   1:  PR[91,3] = PR[90,3] + 136.116;
   1:L PR[91] R[100]mm/sec CNT100;
   1:  PR[91,1] = PR[90,1] + 83.828;
   1:  PR[91,2] = PR[90,2] + 8.492;
   1:  PR[91,3] = PR[90,3] + 136.123;
   1:L PR[91] R[100]mm/sec CNT100;
   1:  PR[91,1] = PR[90,1] + 81.539;
   1:  PR[91,2] = PR[90,2] + 13.617;
   1:  PR[91,3] = PR[90,3] + 136.131;
   1:L PR[91] R[100]mm/sec CNT100;
   1:  PR[91,1] = PR[90,1] + 80.801;
   1:  PR[91,2] = PR[90,2] + 14.808;
   1:  PR[91,3] = PR[90,3] + 136.163;
   1:L PR[91] R[100]mm/sec CNT100;
   1:  PR[91,1] = PR[90,1] + 75.916;
   1:  PR[91,2] = PR[90,2] + 20.688;
   1:  PR[91,3] = PR[90,3] + 136.171;
   1:L PR[91] R[100]mm/sec CNT100;
   1:  PR[91,1] = PR[90,1] + 74.686;
   1:  PR[91,2] = PR[90,2] + 21.792;
   1:  PR[91,3] = PR[90,3] + 136.214;
   1:L PR[91] R[100]mm/sec CNT100;
   1:  PR[91,1] = PR[90,1] + 72.953;
   1:  PR[91,2] = PR[90,2] + 22.987;
   1:  PR[91,3] = PR[90,3] + 136.223;
   1:L PR[91] R[100]mm/sec CNT100;
   1:  PR[91,1] = PR[90,1] + 67.912;
   1:  PR[91,2] = PR[90,2] + 26.567;
   1:  PR[91,3] = PR[90,3] + 136.235;
   1:L PR[91] R[100]mm/sec CNT100;
   1:  PR[91,1] = PR[90,1] + 66.099;
   1:  PR[91,2] = PR[90,2] + 27.495;
   1:  PR[91,3] = PR[90,3] + 136.270;
   1:L PR[91] R[100]mm/sec CNT100;
   1:  PR[91,1] = PR[90,1] + 63.634;
   1:  PR[91,2] = PR[90,2] + 28.417;
   1:  PR[91,3] = PR[90,3] + 136.281;
   1:L PR[91] R[100]mm/sec CNT100;
   1:  PR[91,1] = PR[90,1] + 57.996;
   1:  PR[91,2] = PR[90,2] + 30.575;
   1:  PR[91,3] = PR[90,3] + 136.296;
   1:L PR[91] R[100]mm/sec CNT100;
   1:  PR[91,1] = PR[90,1] + 55.467;
   1:  PR[91,2] = PR[90,2] + 31.181;
   1:  PR[91,3] = PR[90,3] + 136.330;
   1:L PR[91] R[100]mm/sec CNT100;
   1:  PR[91,1] = PR[90,1] + 52.680;
   1:  PR[91,2] = PR[90,2] + 31.695;
   1:  PR[91,3] = PR[90,3] + 136.345;
   1:L PR[91] R[100]mm/sec CNT100;
   1:  PR[91,1] = PR[90,1] + 49.741;
   1:  PR[91,2] = PR[90,2] + 32.053;
   1:  PR[91,3] = PR[90,3] + 136.361;
   1:L PR[91] R[100]mm/sec CNT100;
   1:  PR[91,1] = PR[90,1] + 47.228;
   1:  PR[91,2] = PR[90,2] + 32.206;
   1:  PR[91,3] = PR[90,3] + 136.378;
   1:L PR[91] R[100]mm/sec CNT100;
   1:  PR[91,1] = PR[90,1] + 43.917;
   1:  PR[91,2] = PR[90,2] + 32.236;
   1:  PR[91,3] = PR[90,3] + 136.392;
   1:L PR[91] R[100]mm/sec CNT100;
   1:  PR[91,1] = PR[90,1] + 41.866;
   1:  PR[91,2] = PR[90,2] + 32.111;
   1:  PR[91,3] = PR[90,3] + 136.411;
   1:L PR[91] R[100]mm/sec CNT100;
   1:  PR[91,1] = PR[90,1] + 38.413;
   1:  PR[91,2] = PR[90,2] + 31.768;
   1:  PR[91,3] = PR[90,3] + 136.422;
   1:L PR[91] R[100]mm/sec CNT100;
   1:  PR[91,1] = PR[90,1] + 36.971;
   1:  PR[91,2] = PR[90,2] + 31.502;
   1:  PR[91,3] = PR[90,3] + 136.442;
   1:L PR[91] R[100]mm/sec CNT100;
   1:  PR[91,1] = PR[90,1] + 33.194;
   1:  PR[91,2] = PR[90,2] + 30.719;
   1:  PR[91,3] = PR[90,3] + 136.450;
   1:L PR[91] R[100]mm/sec CNT100;
   1:  PR[91,1] = PR[90,1] + 28.411;
   1:  PR[91,2] = PR[90,2] + 29.184;
   1:  PR[91,3] = PR[90,3] + 136.472;
   1:L PR[91] R[100]mm/sec CNT100;
   1:  PR[91,1] = PR[90,1] + 24.182;
   1:  PR[91,2] = PR[90,2] + 27.259;
   1:  PR[91,3] = PR[90,3] + 136.500;
   1:L PR[91] R[100]mm/sec CNT100;
   1:  PR[91,1] = PR[90,1] + 19.400;
   1:  PR[91,2] = PR[90,2] + 24.371;
   1:  PR[91,3] = PR[90,3] + 136.527;
   1:L PR[91] R[100]mm/sec CNT100;
   1:  PR[91,1] = PR[90,1] + 18.294;
   1:  PR[91,2] = PR[90,2] + 23.512;
   1:  PR[91,3] = PR[90,3] + 136.558;
   1:L PR[91] R[100]mm/sec CNT100;
   1:  PR[91,1] = PR[90,1] + 14.337;
   1:  PR[91,2] = PR[90,2] + 20.137;
   1:  PR[91,3] = PR[90,3] + 136.566;
   1:L PR[91] R[100]mm/sec CNT100;
   1:  PR[91,1] = PR[90,1] + 10.437;
   1:  PR[91,2] = PR[90,2] + 15.629;
   1:  PR[91,3] = PR[90,3] + 136.595;
   1:L PR[91] R[100]mm/sec CNT100;
   1:  PR[91,1] = PR[90,1] + 8.817;
   1:  PR[91,2] = PR[90,2] + 12.942;
   1:  PR[91,3] = PR[90,3] + 136.629;
   1:L PR[91] R[100]mm/sec CNT100;
   1:  PR[91,1] = PR[90,1] + 7.454;
   1:  PR[91,2] = PR[90,2] + 10.581;
   1:  PR[91,3] = PR[90,3] + 136.647;
   1:L PR[91] R[100]mm/sec CNT100;
   1:  PR[91,1] = PR[90,1] + 5.830;
   1:  PR[91,2] = PR[90,2] + 5.883;
   1:  PR[91,3] = PR[90,3] + 136.662;
   1:L PR[91] R[100]mm/sec CNT100;
   1:  PR[91,1] = PR[90,1] + 5.557;
   1:  PR[91,2] = PR[90,2] + 5.060;
   1:  PR[91,3] = PR[90,3] + 136.690;
   1:L PR[91] R[100]mm/sec CNT100;
   1:  PR[91] = PR[90];
   1:  PR[91,1] = PR[90,1] + 6.034;
   1:  PR[91,2] = PR[90,2] + 1.066;
   1:  PR[91,3] = PR[90,3] + 137.995;
   1:L PR[91] R[100]mm/sec CNT100;
   1:  PR[91,1] = PR[90,1] + 5.903;
   1:  PR[91,2] = PR[90,2] + -0.687;
   1:  PR[91,3] = PR[90,3] + 136.717;
   1:L PR[91] R[100]mm/sec CNT100;
   1:  PR[91,1] = PR[90,1] + 6.070;
   1:  PR[91,2] = PR[90,2] + -2.112;
   1:  PR[91,3] = PR[90,3] + 136.727;
   1:L PR[91] R[100]mm/sec CNT100;
   1:  PR[91,1] = PR[90,1] + 6.290;
   1:  PR[91,2] = PR[90,2] + -4.587;
   1:  PR[91,3] = PR[90,3] + 136.735;
   1:L PR[91] R[100]mm/sec CNT100;
   1:  PR[91,1] = PR[90,1] + 6.492;
   1:  PR[91,2] = PR[90,2] + -6.475;
   1:  PR[91,3] = PR[90,3] + 136.749;
   1:L PR[91] R[100]mm/sec CNT100;
   1:  PR[91,1] = PR[90,1] + 7.257;
   1:  PR[91,2] = PR[90,2] + -8.786;
   1:  PR[91,3] = PR[90,3] + 136.760;
   1:L PR[91] R[100]mm/sec CNT100;
   1:  PR[91,1] = PR[90,1] + 8.349;
   1:  PR[91,2] = PR[90,2] + -11.947;
   1:  PR[91,3] = PR[90,3] + 136.774;
   1:L PR[91] R[100]mm/sec CNT100;
   1:  PR[91,1] = PR[90,1] + 10.575;
   1:  PR[91,2] = PR[90,2] + -15.804;
   1:  PR[91,3] = PR[90,3] + 136.793;
   1:L PR[91] R[100]mm/sec CNT100;
   1:  PR[91,1] = PR[90,1] + 11.282;
   1:  PR[91,2] = PR[90,2] + -16.976;
   1:  PR[91,3] = PR[90,3] + 136.818;
   1:L PR[91] R[100]mm/sec CNT100;
   1:  PR[91,1] = PR[90,1] + 13.229;
   1:  PR[91,2] = PR[90,2] + -19.231;
   1:  PR[91,3] = PR[90,3] + 136.826;
   1:L PR[91] R[100]mm/sec CNT100;
   1:  PR[91,1] = PR[90,1] + 15.024;
   1:  PR[91,2] = PR[90,2] + -21.414;
   1:  PR[91,3] = PR[90,3] + 136.843;
   1:L PR[91] R[100]mm/sec CNT100;
   1:  PR[91,1] = PR[90,1] + 15.491;
   1:  PR[91,2] = PR[90,2] + -21.879;
   1:  PR[91,3] = PR[90,3] + 136.858;
   1:L PR[91] R[100]mm/sec CNT100;
   1:  PR[91,1] = PR[90,1] + 18.681;
   1:  PR[91,2] = PR[90,2] + -24.609;
   1:  PR[91,3] = PR[90,3] + 136.862;
   1:L PR[91] R[100]mm/sec CNT100;
   1:  PR[91,1] = PR[90,1] + 20.378;
   1:  PR[91,2] = PR[90,2] + -25.927;
   1:  PR[91,3] = PR[90,3] + 136.886;
   1:L PR[91] R[100]mm/sec CNT100;
   1:  PR[91,1] = PR[90,1] + 22.117;
   1:  PR[91,2] = PR[90,2] + -26.965;
   1:  PR[91,3] = PR[90,3] + 136.898;
   1:L PR[91] R[100]mm/sec CNT100;
   1:  PR[91,1] = PR[90,1] + 24.901;
   1:  PR[91,2] = PR[90,2] + -28.668;
   1:  PR[91,3] = PR[90,3] + 136.909;
   1:L PR[91] R[100]mm/sec CNT100;
   1:  PR[91,1] = PR[90,1] + 28.747;
   1:  PR[91,2] = PR[90,2] + -30.406;
   1:  PR[91,3] = PR[90,3] + 136.928;
   1:L PR[91] R[100]mm/sec CNT100;
   1:  PR[91,1] = PR[90,1] + 31.797;
   1:  PR[91,2] = PR[90,2] + -31.291;
   1:  PR[91,3] = PR[90,3] + 136.952;
   1:L PR[91] R[100]mm/sec CNT100;
   1:  PR[91,1] = PR[90,1] + 34.180;
   1:  PR[91,2] = PR[90,2] + -32.203;
   1:  PR[91,3] = PR[90,3] + 136.970;
   1:L PR[91] R[100]mm/sec CNT100;
   1:  PR[91,1] = PR[90,1] + 37.512;
   1:  PR[91,2] = PR[90,2] + -32.893;
   1:  PR[91,3] = PR[90,3] + 136.984;
   1:L PR[91] R[100]mm/sec CNT100;
   1:  PR[91,1] = PR[90,1] + 39.398;
   1:  PR[91,2] = PR[90,2] + -33.241;
   1:  PR[91,3] = PR[90,3] + 137.003;
   1:L PR[91] R[100]mm/sec CNT100;
   1:  PR[91,1] = PR[90,1] + 42.493;
   1:  PR[91,2] = PR[90,2] + -33.549;
   1:  PR[91,3] = PR[90,3] + 137.014;
   1:L PR[91] R[100]mm/sec CNT100;
   1:  PR[91,1] = PR[90,1] + 44.945;
   1:  PR[91,2] = PR[90,2] + -33.699;
   1:  PR[91,3] = PR[90,3] + 137.032;
   1:L PR[91] R[100]mm/sec CNT100;
   1:  PR[91,1] = PR[90,1] + 47.912;
   1:  PR[91,2] = PR[90,2] + -33.672;
   1:  PR[91,3] = PR[90,3] + 137.046;
   1:L PR[91] R[100]mm/sec CNT100;
   1:  PR[91,1] = PR[90,1] + 50.781;
   1:  PR[91,2] = PR[90,2] + -33.496;
   1:  PR[91,3] = PR[90,3] + 137.062;
   1:L PR[91] R[100]mm/sec CNT100;
   1:  PR[91,1] = PR[90,1] + 53.413;
   1:  PR[91,2] = PR[90,2] + -33.175;
   1:  PR[91,3] = PR[90,3] + 137.079;
   1:L PR[91] R[100]mm/sec CNT100;
   1:  PR[91,1] = PR[90,1] + 56.507;
   1:  PR[91,2] = PR[90,2] + -32.604;
   1:  PR[91,3] = PR[90,3] + 137.094;
   1:L PR[91] R[100]mm/sec CNT100;
   1:  PR[91,1] = PR[90,1] + 58.774;
   1:  PR[91,2] = PR[90,2] + -32.061;
   1:  PR[91,3] = PR[90,3] + 137.111;
   1:L PR[91] R[100]mm/sec CNT100;
   1:  PR[91,1] = PR[90,1] + 60.594;
   1:  PR[91,2] = PR[90,2] + -31.384;
   1:  PR[91,3] = PR[90,3] + 137.124;
   1:L PR[91] R[100]mm/sec CNT100;
   1:  PR[91,1] = PR[90,1] + 67.110;
   1:  PR[91,2] = PR[90,2] + -28.889;
   1:  PR[91,3] = PR[90,3] + 137.135;
   1:L PR[91] R[100]mm/sec CNT100;
   1:  PR[91,1] = PR[90,1] + 68.740;
   1:  PR[91,2] = PR[90,2] + -28.055;
   1:  PR[91,3] = PR[90,3] + 137.175;
   1:L PR[91] R[100]mm/sec CNT100;
   1:  PR[91,1] = PR[90,1] + 70.080;
   1:  PR[91,2] = PR[90,2] + -27.134;
   1:  PR[91,3] = PR[90,3] + 137.185;
   1:L PR[91] R[100]mm/sec CNT100;
   1:  PR[91,1] = PR[90,1] + 75.649;
   1:  PR[91,2] = PR[90,2] + -23.178;
   1:  PR[91,3] = PR[90,3] + 137.194;
   1:L PR[91] R[100]mm/sec CNT100;
   1:  PR[91,1] = PR[90,1] + 76.745;
   1:  PR[91,2] = PR[90,2] + -22.194;
   1:  PR[91,3] = PR[90,3] + 137.233;
   1:L PR[91] R[100]mm/sec CNT100;
   1:  PR[91,1] = PR[90,1] + 81.726;
   1:  PR[91,2] = PR[90,2] + -16.195;
   1:  PR[91,3] = PR[90,3] + 137.241;
   1:L PR[91] R[100]mm/sec CNT100;
   1:  PR[91,1] = PR[90,1] + 82.365;
   1:  PR[91,2] = PR[90,2] + -15.164;
   1:  PR[91,3] = PR[90,3] + 137.285;
   1:L PR[91] R[100]mm/sec CNT100;
   1:  PR[91,1] = PR[90,1] + 82.859;
   1:  PR[91,2] = PR[90,2] + -13.996;
   1:  PR[91,3] = PR[90,3] + 137.292;
   1:L PR[91] R[100]mm/sec CNT100;
   1:  PR[91,1] = PR[90,1] + 85.287;
   1:  PR[91,2] = PR[90,2] + -8.560;
   1:  PR[91,3] = PR[90,3] + 137.299;
   1:L PR[91] R[100]mm/sec CNT100;
   1:  PR[91,1] = PR[90,1] + 85.539;
   1:  PR[91,2] = PR[90,2] + -7.546;
   1:  PR[91,3] = PR[90,3] + 137.333;
   1:L PR[91] R[100]mm/sec CNT100;
   1:  PR[91,1] = PR[90,1] + 85.641;
   1:  PR[91,2] = PR[90,2] + -6.296;
   1:  PR[91,3] = PR[90,3] + 137.339;
   1:L PR[91] R[100]mm/sec CNT100;
   1:  PR[91,1] = PR[90,1] + 86.439;
   1:  PR[91,2] = PR[90,2] + -0.670;
   1:  PR[91,3] = PR[90,3] + 137.346;
   1:L PR[91] R[100]mm/sec CNT100;
   1:  PR[91,1] = PR[90,1] + 86.350;
   1:  PR[91,2] = PR[90,2] + 0.412;
   1:  PR[91,3] = PR[90,3] + 137.378;
   1:L PR[91] R[100]mm/sec CNT100;
   1:  PR[91,1] = PR[90,1] + 85.554;
   1:  PR[91,2] = PR[90,2] + 6.030;
   1:  PR[91,3] = PR[90,3] + 137.384;
   1:L PR[91] R[100]mm/sec CNT100;
   1:  PR[91,1] = PR[90,1] + 85.282;
   1:  PR[91,2] = PR[90,2] + 7.121;
   1:  PR[91,3] = PR[90,3] + 137.416;
   1:L PR[91] R[100]mm/sec CNT100;
   1:  PR[91,1] = PR[90,1] + 84.781;
   1:  PR[91,2] = PR[90,2] + 8.302;
   1:  PR[91,3] = PR[90,3] + 137.422;
   1:L PR[91] R[100]mm/sec CNT100;
   1:  PR[91,1] = PR[90,1] + 82.374;
   1:  PR[91,2] = PR[90,2] + 13.690;
   1:  PR[91,3] = PR[90,3] + 137.430;
   1:L PR[91] R[100]mm/sec CNT100;
   1:  PR[91,1] = PR[90,1] + 81.725;
   1:  PR[91,2] = PR[90,2] + 14.738;
   1:  PR[91,3] = PR[90,3] + 137.463;
   1:L PR[91] R[100]mm/sec CNT100;
   1:  PR[91,1] = PR[90,1] + 76.743;
   1:  PR[91,2] = PR[90,2] + 20.737;
   1:  PR[91,3] = PR[90,3] + 137.470;
   1:L PR[91] R[100]mm/sec CNT100;
   1:  PR[91,1] = PR[90,1] + 75.657;
   1:  PR[91,2] = PR[90,2] + 21.711;
   1:  PR[91,3] = PR[90,3] + 137.514;
   1:L PR[91] R[100]mm/sec CNT100;
   1:  PR[91,1] = PR[90,1] + 74.107;
   1:  PR[91,2] = PR[90,2] + 22.780;
   1:  PR[91,3] = PR[90,3] + 137.522;
   1:L PR[91] R[100]mm/sec CNT100;
   1:  PR[91,1] = PR[90,1] + 68.723;
   1:  PR[91,2] = PR[90,2] + 26.605;
   1:  PR[91,3] = PR[90,3] + 137.533;
   1:L PR[91] R[100]mm/sec CNT100;
   1:  PR[91,1] = PR[90,1] + 67.114;
   1:  PR[91,2] = PR[90,2] + 27.428;
   1:  PR[91,3] = PR[90,3] + 137.570;
   1:L PR[91] R[100]mm/sec CNT100;
   1:  PR[91,1] = PR[90,1] + 64.907;
   1:  PR[91,2] = PR[90,2] + 28.253;
   1:  PR[91,3] = PR[90,3] + 137.580;
   1:L PR[91] R[100]mm/sec CNT100;
   1:  PR[91,1] = PR[90,1] + 58.762;
   1:  PR[91,2] = PR[90,2] + 30.605;
   1:  PR[91,3] = PR[90,3] + 137.594;
   1:L PR[91] R[100]mm/sec CNT100;
   1:  PR[91,1] = PR[90,1] + 56.504;
   1:  PR[91,2] = PR[90,2] + 31.146;
   1:  PR[91,3] = PR[90,3] + 137.631;
   1:L PR[91] R[100]mm/sec CNT100;
   1:  PR[91,1] = PR[90,1] + 53.410;
   1:  PR[91,2] = PR[90,2] + 31.717;
   1:  PR[91,3] = PR[90,3] + 137.644;
   1:L PR[91] R[100]mm/sec CNT100;
   1:  PR[91,1] = PR[90,1] + 50.778;
   1:  PR[91,2] = PR[90,2] + 32.037;
   1:  PR[91,3] = PR[90,3] + 137.662;
   1:L PR[91] R[100]mm/sec CNT100;
   1:  PR[91,1] = PR[90,1] + 47.909;
   1:  PR[91,2] = PR[90,2] + 32.213;
   1:  PR[91,3] = PR[90,3] + 137.677;
   1:L PR[91] R[100]mm/sec CNT100;
   1:  PR[91,1] = PR[90,1] + 44.943;
   1:  PR[91,2] = PR[90,2] + 32.240;
   1:  PR[91,3] = PR[90,3] + 137.693;
   1:L PR[91] R[100]mm/sec CNT100;
   1:  PR[91,1] = PR[90,1] + 42.490;
   1:  PR[91,2] = PR[90,2] + 32.090;
   1:  PR[91,3] = PR[90,3] + 137.710;
   1:L PR[91] R[100]mm/sec CNT100;
   1:  PR[91,1] = PR[90,1] + 39.396;
   1:  PR[91,2] = PR[90,2] + 31.782;
   1:  PR[91,3] = PR[90,3] + 137.724;
   1:L PR[91] R[100]mm/sec CNT100;
   1:  PR[91,1] = PR[90,1] + 37.510;
   1:  PR[91,2] = PR[90,2] + 31.434;
   1:  PR[91,3] = PR[90,3] + 137.741;
   1:L PR[91] R[100]mm/sec CNT100;
   1:  PR[91,1] = PR[90,1] + 34.124;
   1:  PR[91,2] = PR[90,2] + 30.732;
   1:  PR[91,3] = PR[90,3] + 137.752;
   1:L PR[91] R[100]mm/sec CNT100;
   1:  PR[91,1] = PR[90,1] + 29.707;
   1:  PR[91,2] = PR[90,2] + 29.318;
   1:  PR[91,3] = PR[90,3] + 137.771;
   1:L PR[91] R[100]mm/sec CNT100;
   1:  PR[91,1] = PR[90,1] + 26.882;
   1:  PR[91,2] = PR[90,2] + 28.114;
   1:  PR[91,3] = PR[90,3] + 137.798;
   1:L PR[91] R[100]mm/sec CNT100;
   1:  PR[91,1] = PR[90,1] + 24.902;
   1:  PR[91,2] = PR[90,2] + 27.210;
   1:  PR[91,3] = PR[90,3] + 137.815;
   1:L PR[91] R[100]mm/sec CNT100;
   1:  PR[91,1] = PR[90,1] + 20.385;
   1:  PR[91,2] = PR[90,2] + 24.473;
   1:  PR[91,3] = PR[90,3] + 137.827;
   1:L PR[91] R[100]mm/sec CNT100;
   1:  PR[91,1] = PR[90,1] + 18.684;
   1:  PR[91,2] = PR[90,2] + 23.151;
   1:  PR[91,3] = PR[90,3] + 137.857;
   1:L PR[91] R[100]mm/sec CNT100;
   1:  PR[91,1] = PR[90,1] + 15.494;
   1:  PR[91,2] = PR[90,2] + 20.423;
   1:  PR[91,3] = PR[90,3] + 137.869;
   1:L PR[91] R[100]mm/sec CNT100;
   1:  PR[91,1] = PR[90,1] + 15.026;
   1:  PR[91,2] = PR[90,2] + 19.958;
   1:  PR[91,3] = PR[90,3] + 137.893;
   1:L PR[91] R[100]mm/sec CNT100;
   1:  PR[91,1] = PR[90,1] + 13.229;
   1:  PR[91,2] = PR[90,2] + 17.772;
   1:  PR[91,3] = PR[90,3] + 137.897;
   1:L PR[91] R[100]mm/sec CNT100;
   1:  PR[91,1] = PR[90,1] + 11.284;
   1:  PR[91,2] = PR[90,2] + 15.520;
   1:  PR[91,3] = PR[90,3] + 137.913;
   1:L PR[91] R[100]mm/sec CNT100;
   1:  PR[91,1] = PR[90,1] + 10.578;
   1:  PR[91,2] = PR[90,2] + 14.349;
   1:  PR[91,3] = PR[90,3] + 137.929;
   1:L PR[91] R[100]mm/sec CNT100;
   1:  PR[91,1] = PR[90,1] + 8.351;
   1:  PR[91,2] = PR[90,2] + 10.491;
   1:  PR[91,3] = PR[90,3] + 137.937;
   1:L PR[91] R[100]mm/sec CNT100;
   1:  PR[91,1] = PR[90,1] + 7.258;
   1:  PR[91,2] = PR[90,2] + 7.330;
   1:  PR[91,3] = PR[90,3] + 137.962;
   1:L PR[91] R[100]mm/sec CNT100;
   1:  PR[91,1] = PR[90,1] + 6.489;
   1:  PR[91,2] = PR[90,2] + 5.009;
   1:  PR[91,3] = PR[90,3] + 137.981;
   1:L PR[91] R[100]mm/sec CNT100;
   1:  PR[91] = PR[90];
   1:  PR[91,1] = PR[90,1] + 7.128;
   1:  PR[91,2] = PR[90,2] + 2.420;
   1:  PR[91,3] = PR[90,3] + 139.295;
   1:L PR[91] R[100]mm/sec CNT100;
   1:  PR[91,1] = PR[90,1] + 6.959;
   1:  PR[91,2] = PR[90,2] + 0.156;
   1:  PR[91,3] = PR[90,3] + 138.009;
   1:L PR[91] R[100]mm/sec CNT100;
   1:  PR[91,1] = PR[90,1] + 6.863;
   1:  PR[91,2] = PR[90,2] + -0.747;
   1:  PR[91,3] = PR[90,3] + 138.022;
   1:L PR[91] R[100]mm/sec CNT100;
   1:  PR[91,1] = PR[90,1] + 7.088;
   1:  PR[91,2] = PR[90,2] + -3.281;
   1:  PR[91,3] = PR[90,3] + 138.027;
   1:L PR[91] R[100]mm/sec CNT100;
   1:  PR[91,1] = PR[90,1] + 7.424;
   1:  PR[91,2] = PR[90,2] + -6.424;
   1:  PR[91,3] = PR[90,3] + 138.042;
   1:L PR[91] R[100]mm/sec CNT100;
   1:  PR[91,1] = PR[90,1] + 8.684;
   1:  PR[91,2] = PR[90,2] + -10.233;
   1:  PR[91,3] = PR[90,3] + 138.060;
   1:L PR[91] R[100]mm/sec CNT100;
   1:  PR[91,1] = PR[90,1] + 9.246;
   1:  PR[91,2] = PR[90,2] + -11.859;
   1:  PR[91,3] = PR[90,3] + 138.082;
   1:L PR[91] R[100]mm/sec CNT100;
   1:  PR[91,1] = PR[90,1] + 12.150;
   1:  PR[91,2] = PR[90,2] + -16.909;
   1:  PR[91,3] = PR[90,3] + 138.092;
   1:L PR[91] R[100]mm/sec CNT100;
   1:  PR[91,1] = PR[90,1] + 15.624;
   1:  PR[91,2] = PR[90,2] + -21.142;
   1:  PR[91,3] = PR[90,3] + 138.125;
   1:L PR[91] R[100]mm/sec CNT100;
   1:  PR[91,1] = PR[90,1] + 16.758;
   1:  PR[91,2] = PR[90,2] + -22.269;
   1:  PR[91,3] = PR[90,3] + 138.156;
   1:L PR[91] R[100]mm/sec CNT100;
   1:  PR[91,1] = PR[90,1] + 19.070;
   1:  PR[91,2] = PR[90,2] + -24.247;
   1:  PR[91,3] = PR[90,3] + 138.165;
   1:L PR[91] R[100]mm/sec CNT100;
   1:  PR[91,1] = PR[90,1] + 21.369;
   1:  PR[91,2] = PR[90,2] + -26.033;
   1:  PR[91,3] = PR[90,3] + 138.182;
   1:L PR[91] R[100]mm/sec CNT100;
   1:  PR[91,1] = PR[90,1] + 25.631;
   1:  PR[91,2] = PR[90,2] + -28.617;
   1:  PR[91,3] = PR[90,3] + 138.198;
   1:L PR[91] R[100]mm/sec CNT100;
   1:  PR[91,1] = PR[90,1] + 29.090;
   1:  PR[91,2] = PR[90,2] + -30.163;
   1:  PR[91,3] = PR[90,3] + 138.227;
   1:L PR[91] R[100]mm/sec CNT100;
   1:  PR[91,1] = PR[90,1] + 31.798;
   1:  PR[91,2] = PR[90,2] + -30.948;
   1:  PR[91,3] = PR[90,3] + 138.248;
   1:L PR[91] R[100]mm/sec CNT100;
   1:  PR[91,1] = PR[90,1] + 35.111;
   1:  PR[91,2] = PR[90,2] + -32.217;
   1:  PR[91,3] = PR[90,3] + 138.264;
   1:L PR[91] R[100]mm/sec CNT100;
   1:  PR[91,1] = PR[90,1] + 38.052;
   1:  PR[91,2] = PR[90,2] + -32.826;
   1:  PR[91,3] = PR[90,3] + 138.284;
   1:L PR[91] R[100]mm/sec CNT100;
   1:  PR[91,1] = PR[90,1] + 40.381;
   1:  PR[91,2] = PR[90,2] + -33.256;
   1:  PR[91,3] = PR[90,3] + 138.301;
   1:L PR[91] R[100]mm/sec CNT100;
   1:  PR[91,1] = PR[90,1] + 43.117;
   1:  PR[91,2] = PR[90,2] + -33.527;
   1:  PR[91,3] = PR[90,3] + 138.314;
   1:L PR[91] R[100]mm/sec CNT100;
   1:  PR[91,1] = PR[90,1] + 45.972;
   1:  PR[91,2] = PR[90,2] + -33.702;
   1:  PR[91,3] = PR[90,3] + 138.330;
   1:L PR[91] R[100]mm/sec CNT100;
   1:  PR[91,1] = PR[90,1] + 48.594;
   1:  PR[91,2] = PR[90,2] + -33.678;
   1:  PR[91,3] = PR[90,3] + 138.346;
   1:L PR[91] R[100]mm/sec CNT100;
   1:  PR[91,1] = PR[90,1] + 51.818;
   1:  PR[91,2] = PR[90,2] + -33.481;
   1:  PR[91,3] = PR[90,3] + 138.361;
   1:L PR[91] R[100]mm/sec CNT100;
   1:  PR[91,1] = PR[90,1] + 54.143;
   1:  PR[91,2] = PR[90,2] + -33.197;
   1:  PR[91,3] = PR[90,3] + 138.379;
   1:L PR[91] R[100]mm/sec CNT100;
   1:  PR[91,1] = PR[90,1] + 57.546;
   1:  PR[91,2] = PR[90,2] + -32.569;
   1:  PR[91,3] = PR[90,3] + 138.392;
   1:L PR[91] R[100]mm/sec CNT100;
   1:  PR[91,1] = PR[90,1] + 59.541;
   1:  PR[91,2] = PR[90,2] + -32.092;
   1:  PR[91,3] = PR[90,3] + 138.412;
   1:L PR[91] R[100]mm/sec CNT100;
   1:  PR[91,1] = PR[90,1] + 61.144;
   1:  PR[91,2] = PR[90,2] + -31.495;
   1:  PR[91,3] = PR[90,3] + 138.423;
   1:L PR[91] R[100]mm/sec CNT100;
   1:  PR[91,1] = PR[90,1] + 68.125;
   1:  PR[91,2] = PR[90,2] + -28.821;
   1:  PR[91,3] = PR[90,3] + 138.433;
   1:L PR[91] R[100]mm/sec CNT100;
   1:  PR[91,1] = PR[90,1] + 69.550;
   1:  PR[91,2] = PR[90,2] + -28.092;
   1:  PR[91,3] = PR[90,3] + 138.475;
   1:L PR[91] R[100]mm/sec CNT100;
   1:  PR[91,1] = PR[90,1] + 70.728;
   1:  PR[91,2] = PR[90,2] + -27.283;
   1:  PR[91,3] = PR[90,3] + 138.484;
   1:L PR[91] R[100]mm/sec CNT100;
   1:  PR[91,1] = PR[90,1] + 76.620;
   1:  PR[91,2] = PR[90,2] + -23.097;
   1:  PR[91,3] = PR[90,3] + 138.492;
   1:L PR[91] R[100]mm/sec CNT100;
   1:  PR[91,1] = PR[90,1] + 77.572;
   1:  PR[91,2] = PR[90,2] + -22.243;
   1:  PR[91,3] = PR[90,3] + 138.533;
   1:L PR[91] R[100]mm/sec CNT100;
   1:  PR[91,1] = PR[90,1] + 82.650;
   1:  PR[91,2] = PR[90,2] + -16.125;
   1:  PR[91,3] = PR[90,3] + 138.540;
   1:L PR[91] R[100]mm/sec CNT100;
   1:  PR[91,1] = PR[90,1] + 83.201;
   1:  PR[91,2] = PR[90,2] + -15.236;
   1:  PR[91,3] = PR[90,3] + 138.585;
   1:L PR[91] R[100]mm/sec CNT100;
   1:  PR[91,1] = PR[90,1] + 83.634;
   1:  PR[91,2] = PR[90,2] + -14.212;
   1:  PR[91,3] = PR[90,3] + 138.591;
   1:L PR[91] R[100]mm/sec CNT100;
   1:  PR[91,1] = PR[90,1] + 86.177;
   1:  PR[91,2] = PR[90,2] + -8.520;
   1:  PR[91,3] = PR[90,3] + 138.598;
   1:L PR[91] R[100]mm/sec CNT100;
   1:  PR[91,1] = PR[90,1] + 86.391;
   1:  PR[91,2] = PR[90,2] + -7.655;
   1:  PR[91,3] = PR[90,3] + 138.633;
   1:L PR[91] R[100]mm/sec CNT100;
   1:  PR[91,1] = PR[90,1] + 86.481;
   1:  PR[91,2] = PR[90,2] + -6.556;
   1:  PR[91,3] = PR[90,3] + 138.638;
   1:L PR[91] R[100]mm/sec CNT100;
   1:  PR[91,1] = PR[90,1] + 87.316;
   1:  PR[91,2] = PR[90,2] + -0.670;
   1:  PR[91,3] = PR[90,3] + 138.644;
   1:L PR[91] R[100]mm/sec CNT100;
   1:  PR[91,1] = PR[90,1] + 87.240;
   1:  PR[91,2] = PR[90,2] + 0.260;
   1:  PR[91,3] = PR[90,3] + 138.678;
   1:L PR[91] R[100]mm/sec CNT100;
   1:  PR[91,1] = PR[90,1] + 86.406;
   1:  PR[91,2] = PR[90,2] + 6.139;
   1:  PR[91,3] = PR[90,3] + 138.683;
   1:L PR[91] R[100]mm/sec CNT100;
   1:  PR[91,1] = PR[90,1] + 86.172;
   1:  PR[91,2] = PR[90,2] + 7.080;
   1:  PR[91,3] = PR[90,3] + 138.716;
   1:L PR[91] R[100]mm/sec CNT100;
   1:  PR[91,1] = PR[90,1] + 85.734;
   1:  PR[91,2] = PR[90,2] + 8.112;
   1:  PR[91,3] = PR[90,3] + 138.722;
   1:L PR[91] R[100]mm/sec CNT100;
   1:  PR[91,1] = PR[90,1] + 83.210;
   1:  PR[91,2] = PR[90,2] + 13.762;
   1:  PR[91,3] = PR[90,3] + 138.728;
   1:L PR[91] R[100]mm/sec CNT100;
   1:  PR[91,1] = PR[90,1] + 82.649;
   1:  PR[91,2] = PR[90,2] + 14.667;
   1:  PR[91,3] = PR[90,3] + 138.763;
   1:L PR[91] R[100]mm/sec CNT100;
   1:  PR[91,1] = PR[90,1] + 77.570;
   1:  PR[91,2] = PR[90,2] + 20.786;
   1:  PR[91,3] = PR[90,3] + 138.769;
   1:L PR[91] R[100]mm/sec CNT100;
   1:  PR[91,1] = PR[90,1] + 76.628;
   1:  PR[91,2] = PR[90,2] + 21.631;
   1:  PR[91,3] = PR[90,3] + 138.814;
   1:L PR[91] R[100]mm/sec CNT100;
   1:  PR[91,1] = PR[90,1] + 75.262;
   1:  PR[91,2] = PR[90,2] + 22.573;
   1:  PR[91,3] = PR[90,3] + 138.821;
   1:L PR[91] R[100]mm/sec CNT100;
   1:  PR[91,1] = PR[90,1] + 69.533;
   1:  PR[91,2] = PR[90,2] + 26.642;
   1:  PR[91,3] = PR[90,3] + 138.831;
   1:L PR[91] R[100]mm/sec CNT100;
   1:  PR[91,1] = PR[90,1] + 68.129;
   1:  PR[91,2] = PR[90,2] + 27.360;
   1:  PR[91,3] = PR[90,3] + 138.870;
   1:L PR[91] R[100]mm/sec CNT100;
   1:  PR[91,1] = PR[90,1] + 66.180;
   1:  PR[91,2] = PR[90,2] + 28.089;
   1:  PR[91,3] = PR[90,3] + 138.879;
   1:L PR[91] R[100]mm/sec CNT100;
   1:  PR[91,1] = PR[90,1] + 59.528;
   1:  PR[91,2] = PR[90,2] + 30.636;
   1:  PR[91,3] = PR[90,3] + 138.891;
   1:L PR[91] R[100]mm/sec CNT100;
   1:  PR[91,1] = PR[90,1] + 57.542;
   1:  PR[91,2] = PR[90,2] + 31.111;
   1:  PR[91,3] = PR[90,3] + 138.931;
   1:L PR[91] R[100]mm/sec CNT100;
   1:  PR[91,1] = PR[90,1] + 54.140;
   1:  PR[91,2] = PR[90,2] + 31.739;
   1:  PR[91,3] = PR[90,3] + 138.943;
   1:L PR[91] R[100]mm/sec CNT100;
   1:  PR[91,1] = PR[90,1] + 51.815;
   1:  PR[91,2] = PR[90,2] + 32.022;
   1:  PR[91,3] = PR[90,3] + 138.962;
   1:L PR[91] R[100]mm/sec CNT100;
   1:  PR[91,1] = PR[90,1] + 48.591;
   1:  PR[91,2] = PR[90,2] + 32.219;
   1:  PR[91,3] = PR[90,3] + 138.976;
   1:L PR[91] R[100]mm/sec CNT100;
   1:  PR[91,1] = PR[90,1] + 45.969;
   1:  PR[91,2] = PR[90,2] + 32.243;
   1:  PR[91,3] = PR[90,3] + 138.994;
   1:L PR[91] R[100]mm/sec CNT100;
   1:  PR[91,1] = PR[90,1] + 43.114;
   1:  PR[91,2] = PR[90,2] + 32.068;
   1:  PR[91,3] = PR[90,3] + 139.009;
   1:L PR[91] R[100]mm/sec CNT100;
   1:  PR[91,1] = PR[90,1] + 40.379;
   1:  PR[91,2] = PR[90,2] + 31.797;
   1:  PR[91,3] = PR[90,3] + 139.025;
   1:L PR[91] R[100]mm/sec CNT100;
   1:  PR[91,1] = PR[90,1] + 38.049;
   1:  PR[91,2] = PR[90,2] + 31.366;
   1:  PR[91,3] = PR[90,3] + 139.040;
   1:L PR[91] R[100]mm/sec CNT100;
   1:  PR[91,1] = PR[90,1] + 35.055;
   1:  PR[91,2] = PR[90,2] + 30.746;
   1:  PR[91,3] = PR[90,3] + 139.054;
   1:L PR[91] R[100]mm/sec CNT100;
   1:  PR[91,1] = PR[90,1] + 31.151;
   1:  PR[91,2] = PR[90,2] + 29.496;
   1:  PR[91,3] = PR[90,3] + 139.071;
   1:L PR[91] R[100]mm/sec CNT100;
   1:  PR[91,1] = PR[90,1] + 25.718;
   1:  PR[91,2] = PR[90,2] + 27.181;
   1:  PR[91,3] = PR[90,3] + 139.094;
   1:L PR[91] R[100]mm/sec CNT100;
   1:  PR[91,1] = PR[90,1] + 25.584;
   1:  PR[91,2] = PR[90,2] + 27.130;
   1:  PR[91,3] = PR[90,3] + 139.127;
   1:L PR[91] R[100]mm/sec CNT100;
   1:  PR[91,1] = PR[90,1] + 21.370;
   1:  PR[91,2] = PR[90,2] + 24.575;
   1:  PR[91,3] = PR[90,3] + 139.128;
   1:L PR[91] R[100]mm/sec CNT100;
   1:  PR[91,1] = PR[90,1] + 19.072;
   1:  PR[91,2] = PR[90,2] + 22.789;
   1:  PR[91,3] = PR[90,3] + 139.156;
   1:L PR[91] R[100]mm/sec CNT100;
   1:  PR[91,1] = PR[90,1] + 16.761;
   1:  PR[91,2] = PR[90,2] + 20.813;
   1:  PR[91,3] = PR[90,3] + 139.173;
   1:L PR[91] R[100]mm/sec CNT100;
   1:  PR[91,1] = PR[90,1] + 15.626;
   1:  PR[91,2] = PR[90,2] + 19.685;
   1:  PR[91,3] = PR[90,3] + 139.190;
   1:L PR[91] R[100]mm/sec CNT100;
   1:  PR[91,1] = PR[90,1] + 12.152;
   1:  PR[91,2] = PR[90,2] + 15.452;
   1:  PR[91,3] = PR[90,3] + 139.199;
   1:L PR[91] R[100]mm/sec CNT100;
   1:  PR[91,1] = PR[90,1] + 9.247;
   1:  PR[91,2] = PR[90,2] + 10.402;
   1:  PR[91,3] = PR[90,3] + 139.230;
   1:L PR[91] R[100]mm/sec CNT100;
   1:  PR[91,1] = PR[90,1] + 8.685;
   1:  PR[91,2] = PR[90,2] + 8.776;
   1:  PR[91,3] = PR[90,3] + 139.263;
   1:L PR[91] R[100]mm/sec CNT100;
   1:  PR[91,1] = PR[90,1] + 7.421;
   1:  PR[91,2] = PR[90,2] + 4.958;
   1:  PR[91,3] = PR[90,3] + 139.272;
   1:L PR[91] R[100]mm/sec CNT100;
   1:  PR[91] = PR[90];
   1:  PR[91,1] = PR[90,1] + 8.222;
   1:  PR[91,2] = PR[90,2] + 3.775;
   1:  PR[91,3] = PR[90,3] + 140.595;
   1:L PR[91] R[100]mm/sec CNT100;
   1:  PR[91,1] = PR[90,1] + 8.139;
   1:  PR[91,2] = PR[90,2] + 2.659;
   1:  PR[91,3] = PR[90,3] + 139.301;
   1:L PR[91] R[100]mm/sec CNT100;
   1:  PR[91,1] = PR[90,1] + 7.777;
   1:  PR[91,2] = PR[90,2] + -0.747;
   1:  PR[91,3] = PR[90,3] + 139.308;
   1:L PR[91] R[100]mm/sec CNT100;
   1:  PR[91,1] = PR[90,1] + 7.886;
   1:  PR[91,2] = PR[90,2] + -1.975;
   1:  PR[91,3] = PR[90,3] + 139.327;
   1:L PR[91] R[100]mm/sec CNT100;
   1:  PR[91,1] = PR[90,1] + 8.356;
   1:  PR[91,2] = PR[90,2] + -6.373;
   1:  PR[91,3] = PR[90,3] + 139.334;
   1:L PR[91] R[100]mm/sec CNT100;
   1:  PR[91,1] = PR[90,1] + 10.112;
   1:  PR[91,2] = PR[90,2] + -11.680;
   1:  PR[91,3] = PR[90,3] + 139.359;
   1:L PR[91] R[100]mm/sec CNT100;
   1:  PR[91,1] = PR[90,1] + 10.142;
   1:  PR[91,2] = PR[90,2] + -11.768;
   1:  PR[91,3] = PR[90,3] + 139.391;
   1:L PR[91] R[100]mm/sec CNT100;
   1:  PR[91,1] = PR[90,1] + 10.489;
   1:  PR[91,2] = PR[90,2] + -12.369;
   1:L PR[91] R[100]mm/sec CNT100;
   1:  PR[91,1] = PR[90,1] + 12.986;
   1:  PR[91,2] = PR[90,2] + -16.874;
   1:  PR[91,3] = PR[90,3] + 139.395;
   1:L PR[91] R[100]mm/sec CNT100;
   1:  PR[91,1] = PR[90,1] + 13.647;
   1:  PR[91,2] = PR[90,2] + -17.733;
   1:  PR[91,3] = PR[90,3] + 139.424;
   1:L PR[91] R[100]mm/sec CNT100;
   1:  PR[91,1] = PR[90,1] + 16.224;
   1:  PR[91,2] = PR[90,2] + -20.868;
   1:  PR[91,3] = PR[90,3] + 139.430;
   1:L PR[91] R[100]mm/sec CNT100;
   1:  PR[91,1] = PR[90,1] + 18.025;
   1:  PR[91,2] = PR[90,2] + -22.659;
   1:  PR[91,3] = PR[90,3] + 139.453;
   1:L PR[91] R[100]mm/sec CNT100;
   1:  PR[91,1] = PR[90,1] + 19.459;
   1:  PR[91,2] = PR[90,2] + -23.885;
   1:  PR[91,3] = PR[90,3] + 139.468;
   1:L PR[91] R[100]mm/sec CNT100;
   1:  PR[91,1] = PR[90,1] + 22.350;
   1:  PR[91,2] = PR[90,2] + -26.131;
   1:  PR[91,3] = PR[90,3] + 139.478;
   1:L PR[91] R[100]mm/sec CNT100;
   1:  PR[91,1] = PR[90,1] + 26.437;
   1:  PR[91,2] = PR[90,2] + -28.580;
   1:  PR[91,3] = PR[90,3] + 139.499;
   1:L PR[91] R[100]mm/sec CNT100;
   1:  PR[91,1] = PR[90,1] + 29.437;
   1:  PR[91,2] = PR[90,2] + -29.920;
   1:  PR[91,3] = PR[90,3] + 139.526;
   1:L PR[91] R[100]mm/sec CNT100;
   1:  PR[91,1] = PR[90,1] + 31.798;
   1:  PR[91,2] = PR[90,2] + -30.605;
   1:  PR[91,3] = PR[90,3] + 139.544;
   1:L PR[91] R[100]mm/sec CNT100;
   1:  PR[91,1] = PR[90,1] + 36.042;
   1:  PR[91,2] = PR[90,2] + -32.230;
   1:  PR[91,3] = PR[90,3] + 139.558;
   1:L PR[91] R[100]mm/sec CNT100;
   1:  PR[91,1] = PR[90,1] + 38.591;
   1:  PR[91,2] = PR[90,2] + -32.758;
   1:  PR[91,3] = PR[90,3] + 139.584;
   1:L PR[91] R[100]mm/sec CNT100;
   1:  PR[91,1] = PR[90,1] + 41.365;
   1:  PR[91,2] = PR[90,2] + -33.270;
   1:  PR[91,3] = PR[90,3] + 139.599;
   1:L PR[91] R[100]mm/sec CNT100;
   1:  PR[91,1] = PR[90,1] + 43.742;
   1:  PR[91,2] = PR[90,2] + -33.506;
   1:  PR[91,3] = PR[90,3] + 139.615;
   1:L PR[91] R[100]mm/sec CNT100;
   1:  PR[91,1] = PR[90,1] + 46.998;
   1:  PR[91,2] = PR[90,2] + -33.705;
   1:  PR[91,3] = PR[90,3] + 139.628;
   1:L PR[91] R[100]mm/sec CNT100;
   1:  PR[91,1] = PR[90,1] + 49.276;
   1:  PR[91,2] = PR[90,2] + -33.685;
   1:  PR[91,3] = PR[90,3] + 139.647;
   1:L PR[91] R[100]mm/sec CNT100;
   1:  PR[91,1] = PR[90,1] + 52.855;
   1:  PR[91,2] = PR[90,2] + -33.465;
   1:  PR[91,3] = PR[90,3] + 139.659;
   1:L PR[91] R[100]mm/sec CNT100;
   1:  PR[91,1] = PR[90,1] + 54.873;
   1:  PR[91,2] = PR[90,2] + -33.220;
   1:  PR[91,3] = PR[90,3] + 139.680;
   1:L PR[91] R[100]mm/sec CNT100;
   1:  PR[91,1] = PR[90,1] + 58.584;
   1:  PR[91,2] = PR[90,2] + -32.534;
   1:  PR[91,3] = PR[90,3] + 139.691;
   1:L PR[91] R[100]mm/sec CNT100;
   1:  PR[91,1] = PR[90,1] + 60.307;
   1:  PR[91,2] = PR[90,2] + -32.122;
   1:  PR[91,3] = PR[90,3] + 139.712;
   1:L PR[91] R[100]mm/sec CNT100;
   1:  PR[91,1] = PR[90,1] + 61.693;
   1:  PR[91,2] = PR[90,2] + -31.606;
   1:  PR[91,3] = PR[90,3] + 139.722;
   1:L PR[91] R[100]mm/sec CNT100;
   1:  PR[91,1] = PR[90,1] + 69.141;
   1:  PR[91,2] = PR[90,2] + -28.754;
   1:  PR[91,3] = PR[90,3] + 139.731;
   1:L PR[91] R[100]mm/sec CNT100;
   1:  PR[91,1] = PR[90,1] + 70.361;
   1:  PR[91,2] = PR[90,2] + -28.130;
   1:  PR[91,3] = PR[90,3] + 139.776;
   1:L PR[91] R[100]mm/sec CNT100;
   1:  PR[91,1] = PR[90,1] + 71.375;
   1:  PR[91,2] = PR[90,2] + -27.433;
   1:  PR[91,3] = PR[90,3] + 139.784;
   1:L PR[91] R[100]mm/sec CNT100;
   1:  PR[91,1] = PR[90,1] + 77.591;
   1:  PR[91,2] = PR[90,2] + -23.016;
   1:  PR[91,3] = PR[90,3] + 139.791;
   1:L PR[91] R[100]mm/sec CNT100;
   1:  PR[91,1] = PR[90,1] + 78.399;
   1:  PR[91,2] = PR[90,2] + -22.291;
   1:  PR[91,3] = PR[90,3] + 139.834;
   1:L PR[91] R[100]mm/sec CNT100;
   1:  PR[91,1] = PR[90,1] + 83.574;
   1:  PR[91,2] = PR[90,2] + -16.055;
   1:  PR[91,3] = PR[90,3] + 139.840;
   1:L PR[91] R[100]mm/sec CNT100;
   1:  PR[91,1] = PR[90,1] + 84.036;
   1:  PR[91,2] = PR[90,2] + -15.309;
   1:  PR[91,3] = PR[90,3] + 139.886;
   1:L PR[91] R[100]mm/sec CNT100;
   1:  PR[91,1] = PR[90,1] + 84.409;
   1:  PR[91,2] = PR[90,2] + -14.429;
   1:  PR[91,3] = PR[90,3] + 139.891;
   1:L PR[91] R[100]mm/sec CNT100;
   1:  PR[91,1] = PR[90,1] + 87.066;
   1:  PR[91,2] = PR[90,2] + -8.479;
   1:  PR[91,3] = PR[90,3] + 139.896;
   1:L PR[91] R[100]mm/sec CNT100;
   1:  PR[91,1] = PR[90,1] + 87.244;
   1:  PR[91,2] = PR[90,2] + -7.765;
   1:  PR[91,3] = PR[90,3] + 139.933;
   1:L PR[91] R[100]mm/sec CNT100;
   1:  PR[91,1] = PR[90,1] + 87.321;
   1:  PR[91,2] = PR[90,2] + -6.817;
   1:  PR[91,3] = PR[90,3] + 139.937;
   1:L PR[91] R[100]mm/sec CNT100;
   1:  PR[91,1] = PR[90,1] + 88.193;
   1:  PR[91,2] = PR[90,2] + -0.670;
   1:  PR[91,3] = PR[90,3] + 139.942;
   1:L PR[91] R[100]mm/sec CNT100;
   1:  PR[91,1] = PR[90,1] + 88.129;
   1:  PR[91,2] = PR[90,2] + 0.108;
   1:  PR[91,3] = PR[90,3] + 139.977;
   1:L PR[91] R[100]mm/sec CNT100;
   1:  PR[91,1] = PR[90,1] + 87.258;
   1:  PR[91,2] = PR[90,2] + 6.249;
   1:  PR[91,3] = PR[90,3] + 139.982;
   1:L PR[91] R[100]mm/sec CNT100;
   1:  PR[91,1] = PR[90,1] + 87.061;
   1:  PR[91,2] = PR[90,2] + 7.039;
   1:  PR[91,3] = PR[90,3] + 140.017;
   1:L PR[91] R[100]mm/sec CNT100;
   1:  PR[91,1] = PR[90,1] + 86.687;
   1:  PR[91,2] = PR[90,2] + 7.921;
   1:  PR[91,3] = PR[90,3] + 140.021;
   1:L PR[91] R[100]mm/sec CNT100;
   1:  PR[91,1] = PR[90,1] + 84.046;
   1:  PR[91,2] = PR[90,2] + 13.835;
   1:  PR[91,3] = PR[90,3] + 140.027;
   1:L PR[91] R[100]mm/sec CNT100;
   1:  PR[91,1] = PR[90,1] + 83.573;
   1:  PR[91,2] = PR[90,2] + 14.597;
   1:  PR[91,3] = PR[90,3] + 140.063;
   1:L PR[91] R[100]mm/sec CNT100;
   1:  PR[91,1] = PR[90,1] + 78.397;
   1:  PR[91,2] = PR[90,2] + 20.835;
   1:  PR[91,3] = PR[90,3] + 140.068;
   1:L PR[91] R[100]mm/sec CNT100;
   1:  PR[91,1] = PR[90,1] + 77.599;
   1:  PR[91,2] = PR[90,2] + 21.550;
   1:  PR[91,3] = PR[90,3] + 140.114;
   1:L PR[91] R[100]mm/sec CNT100;
   1:  PR[91,1] = PR[90,1] + 76.416;
   1:  PR[91,2] = PR[90,2] + 22.366;
   1:  PR[91,3] = PR[90,3] + 140.120;
   1:L PR[91] R[100]mm/sec CNT100;
   1:  PR[91,1] = PR[90,1] + 70.343;
   1:  PR[91,2] = PR[90,2] + 26.680;
   1:  PR[91,3] = PR[90,3] + 140.128;
   1:L PR[91] R[100]mm/sec CNT100;
   1:  PR[91,1] = PR[90,1] + 69.145;
   1:  PR[91,2] = PR[90,2] + 27.293;
   1:  PR[91,3] = PR[90,3] + 140.171;
   1:L PR[91] R[100]mm/sec CNT100;
   1:  PR[91,1] = PR[90,1] + 67.452;
   1:  PR[91,2] = PR[90,2] + 27.926;
   1:  PR[91,3] = PR[90,3] + 140.178;
   1:L PR[91] R[100]mm/sec CNT100;
   1:  PR[91,1] = PR[90,1] + 60.294;
   1:  PR[91,2] = PR[90,2] + 30.666;
   1:  PR[91,3] = PR[90,3] + 140.188;
   1:L PR[91] R[100]mm/sec CNT100;
   1:  PR[91,1] = PR[90,1] + 58.580;
   1:  PR[91,2] = PR[90,2] + 31.077;
   1:  PR[91,3] = PR[90,3] + 140.232;
   1:L PR[91] R[100]mm/sec CNT100;
   1:  PR[91,1] = PR[90,1] + 54.869;
   1:  PR[91,2] = PR[90,2] + 31.761;
   1:  PR[91,3] = PR[90,3] + 140.242;
   1:L PR[91] R[100]mm/sec CNT100;
   1:  PR[91,1] = PR[90,1] + 52.851;
   1:  PR[91,2] = PR[90,2] + 32.007;
   1:  PR[91,3] = PR[90,3] + 140.263;
   1:L PR[91] R[100]mm/sec CNT100;
   1:  PR[91,1] = PR[90,1] + 49.273;
   1:  PR[91,2] = PR[90,2] + 32.226;
   1:  PR[91,3] = PR[90,3] + 140.274;
   1:L PR[91] R[100]mm/sec CNT100;
   1:  PR[91,1] = PR[90,1] + 46.995;
   1:  PR[91,2] = PR[90,2] + 32.247;
   1:  PR[91,3] = PR[90,3] + 140.295;
   1:L PR[91] R[100]mm/sec CNT100;
   1:  PR[91,1] = PR[90,1] + 43.739;
   1:  PR[91,2] = PR[90,2] + 32.047;
   1:  PR[91,3] = PR[90,3] + 140.308;
   1:L PR[91] R[100]mm/sec CNT100;
   1:  PR[91,1] = PR[90,1] + 41.362;
   1:  PR[91,2] = PR[90,2] + 31.811;
   1:  PR[91,3] = PR[90,3] + 140.326;
   1:L PR[91] R[100]mm/sec CNT100;
   1:  PR[91,1] = PR[90,1] + 38.589;
   1:  PR[91,2] = PR[90,2] + 31.299;
   1:  PR[91,3] = PR[90,3] + 140.339;
   1:L PR[91] R[100]mm/sec CNT100;
   1:  PR[91,1] = PR[90,1] + 35.985;
   1:  PR[91,2] = PR[90,2] + 30.759;
   1:  PR[91,3] = PR[90,3] + 140.355;
   1:L PR[91] R[100]mm/sec CNT100;
   1:  PR[91,1] = PR[90,1] + 32.596;
   1:  PR[91,2] = PR[90,2] + 29.674;
   1:  PR[91,3] = PR[90,3] + 140.370;
   1:L PR[91] R[100]mm/sec CNT100;
   1:  PR[91,1] = PR[90,1] + 27.851;
   1:  PR[91,2] = PR[90,2] + 27.652;
   1:  PR[91,3] = PR[90,3] + 140.391;
   1:L PR[91] R[100]mm/sec CNT100;
   1:  PR[91,1] = PR[90,1] + 26.389;
   1:  PR[91,2] = PR[90,2] + 27.093;
   1:  PR[91,3] = PR[90,3] + 140.420;
   1:L PR[91] R[100]mm/sec CNT100;
   1:  PR[91,1] = PR[90,1] + 22.351;
   1:  PR[91,2] = PR[90,2] + 24.673;
   1:  PR[91,3] = PR[90,3] + 140.428;
   1:L PR[91] R[100]mm/sec CNT100;
   1:  PR[91,1] = PR[90,1] + 19.460;
   1:  PR[91,2] = PR[90,2] + 22.428;
   1:  PR[91,3] = PR[90,3] + 140.455;
   1:L PR[91] R[100]mm/sec CNT100;
   1:  PR[91,1] = PR[90,1] + 18.027;
   1:  PR[91,2] = PR[90,2] + 21.202;
   1:  PR[91,3] = PR[90,3] + 140.476;
   1:L PR[91] R[100]mm/sec CNT100;
   1:  PR[91,1] = PR[90,1] + 16.226;
   1:  PR[91,2] = PR[90,2] + 19.411;
   1:  PR[91,3] = PR[90,3] + 140.486;
   1:L PR[91] R[100]mm/sec CNT100;
   1:  PR[91,1] = PR[90,1] + 13.649;
   1:  PR[91,2] = PR[90,2] + 16.277;
   1:  PR[91,3] = PR[90,3] + 140.501;
   1:L PR[91] R[100]mm/sec CNT100;
   1:  PR[91,1] = PR[90,1] + 12.988;
   1:  PR[91,2] = PR[90,2] + 15.417;
   1:  PR[91,3] = PR[90,3] + 140.524;
   1:L PR[91] R[100]mm/sec CNT100;
   1:  PR[91,1] = PR[90,1] + 10.489;
   1:  PR[91,2] = PR[90,2] + 10.910;
   1:  PR[91,3] = PR[90,3] + 140.530;
   1:L PR[91] R[100]mm/sec CNT100;
   1:  PR[91,1] = PR[90,1] + 10.149;
   1:  PR[91,2] = PR[90,2] + 10.322;
   1:  PR[91,3] = PR[90,3] + 140.559;
   1:L PR[91] R[100]mm/sec CNT100;
   1:  PR[91,1] = PR[90,1] + 8.353;
   1:  PR[91,2] = PR[90,2] + 4.907;
   1:  PR[91,3] = PR[90,3] + 140.563;
   1:L PR[91] R[100]mm/sec CNT100;
   1:  PR[91] = PR[90];
   1:  PR[91,1] = PR[90,1] + 8.691;
   1:  PR[91,2] = PR[90,2] + -0.740;
   1:  PR[91,3] = PR[90,3] + 141.895;
   1:L PR[91] R[100]mm/sec CNT100;
   1:  PR[91,1] = PR[90,1] + 9.287;
   1:  PR[91,2] = PR[90,2] + -6.332;
   1:  PR[91,3] = PR[90,3] + 140.627;
   1:L PR[91] R[100]mm/sec CNT100;
   1:  PR[91,1] = PR[90,1] + 10.891;
   1:  PR[91,2] = PR[90,2] + -11.428;
   1:  PR[91,3] = PR[90,3] + 140.659;
   1:L PR[91] R[100]mm/sec CNT100;
   1:  PR[91,1] = PR[90,1] + 11.087;
   1:  PR[91,2] = PR[90,2] + -11.925;
   1:  PR[91,3] = PR[90,3] + 140.689;
   1:L PR[91] R[100]mm/sec CNT100;
   1:  PR[91,1] = PR[90,1] + 13.067;
   1:  PR[91,2] = PR[90,2] + -15.512;
   1:  PR[91,3] = PR[90,3] + 140.692;
   1:L PR[91] R[100]mm/sec CNT100;
   1:  PR[91,1] = PR[90,1] + 13.792;
   1:  PR[91,2] = PR[90,2] + -16.792;
   1:  PR[91,3] = PR[90,3] + 140.715;
   1:L PR[91] R[100]mm/sec CNT100;
   1:  PR[91,1] = PR[90,1] + 15.147;
   1:  PR[91,2] = PR[90,2] + -18.555;
   1:  PR[91,3] = PR[90,3] + 140.723;
   1:L PR[91] R[100]mm/sec CNT100;
   1:  PR[91,1] = PR[90,1] + 16.825;
   1:  PR[91,2] = PR[90,2] + -20.595;
   1:  PR[91,3] = PR[90,3] + 140.736;
   1:L PR[91] R[100]mm/sec CNT100;
   1:  PR[91,1] = PR[90,1] + 19.292;
   1:  PR[91,2] = PR[90,2] + -23.049;
   1:  PR[91,3] = PR[90,3] + 140.751;
   1:L PR[91] R[100]mm/sec CNT100;
   1:  PR[91,1] = PR[90,1] + 19.845;
   1:  PR[91,2] = PR[90,2] + -23.521;
   1:  PR[91,3] = PR[90,3] + 140.770;
   1:L PR[91] R[100]mm/sec CNT100;
   1:  PR[91,1] = PR[90,1] + 22.849;
   1:  PR[91,2] = PR[90,2] + -25.836;
   1:  PR[91,3] = PR[90,3] + 140.775;
   1:L PR[91] R[100]mm/sec CNT100;
   1:  PR[91,1] = PR[90,1] + 23.602;
   1:  PR[91,2] = PR[90,2] + -26.371;
   1:  PR[91,3] = PR[90,3] + 140.796;
   1:L PR[91] R[100]mm/sec CNT100;
   1:  PR[91,1] = PR[90,1] + 27.247;
   1:  PR[91,2] = PR[90,2] + -28.545;
   1:  PR[91,3] = PR[90,3] + 140.801;
   1:L PR[91] R[100]mm/sec CNT100;
   1:  PR[91,1] = PR[90,1] + 29.784;
   1:  PR[91,2] = PR[90,2] + -29.678;
   1:  PR[91,3] = PR[90,3] + 140.825;
   1:L PR[91] R[100]mm/sec CNT100;
   1:  PR[91,1] = PR[90,1] + 31.798;
   1:  PR[91,2] = PR[90,2] + -30.263;
   1:  PR[91,3] = PR[90,3] + 140.841;
   1:L PR[91] R[100]mm/sec CNT100;
   1:  PR[91,1] = PR[90,1] + 36.973;
   1:  PR[91,2] = PR[90,2] + -32.244;
   1:  PR[91,3] = PR[90,3] + 140.853;
   1:L PR[91] R[100]mm/sec CNT100;
   1:  PR[91,1] = PR[90,1] + 39.131;
   1:  PR[91,2] = PR[90,2] + -32.691;
   1:  PR[91,3] = PR[90,3] + 140.884;
   1:L PR[91] R[100]mm/sec CNT100;
   1:  PR[91,1] = PR[90,1] + 42.348;
   1:  PR[91,2] = PR[90,2] + -33.285;
   1:  PR[91,3] = PR[90,3] + 140.897;
   1:L PR[91] R[100]mm/sec CNT100;
   1:  PR[91,1] = PR[90,1] + 44.367;
   1:  PR[91,2] = PR[90,2] + -33.485;
   1:  PR[91,3] = PR[90,3] + 140.915;
   1:L PR[91] R[100]mm/sec CNT100;
   1:  PR[91,1] = PR[90,1] + 48.025;
   1:  PR[91,2] = PR[90,2] + -33.709;
   1:  PR[91,3] = PR[90,3] + 140.926;
   1:L PR[91] R[100]mm/sec CNT100;
   1:  PR[91,1] = PR[90,1] + 49.958;
   1:  PR[91,2] = PR[90,2] + -33.691;
   1:  PR[91,3] = PR[90,3] + 140.947;
   1:L PR[91] R[100]mm/sec CNT100;
   1:  PR[91,1] = PR[90,1] + 53.892;
   1:  PR[91,2] = PR[90,2] + -33.450;
   1:  PR[91,3] = PR[90,3] + 140.958;
   1:L PR[91] R[100]mm/sec CNT100;
   1:  PR[91,1] = PR[90,1] + 55.603;
   1:  PR[91,2] = PR[90,2] + -33.242;
   1:  PR[91,3] = PR[90,3] + 140.980;
   1:L PR[91] R[100]mm/sec CNT100;
   1:  PR[91,1] = PR[90,1] + 59.622;
   1:  PR[91,2] = PR[90,2] + -32.500;
   1:  PR[91,3] = PR[90,3] + 140.990;
   1:L PR[91] R[100]mm/sec CNT100;
   1:  PR[91,1] = PR[90,1] + 61.074;
   1:  PR[91,2] = PR[90,2] + -32.152;
   1:  PR[91,3] = PR[90,3] + 141.013;
   1:L PR[91] R[100]mm/sec CNT100;
   1:  PR[91,1] = PR[90,1] + 62.243;
   1:  PR[91,2] = PR[90,2] + -31.717;
   1:  PR[91,3] = PR[90,3] + 141.022;
   1:L PR[91] R[100]mm/sec CNT100;
   1:  PR[91,1] = PR[90,1] + 70.157;
   1:  PR[91,2] = PR[90,2] + -28.686;
   1:  PR[91,3] = PR[90,3] + 141.029;
   1:L PR[91] R[100]mm/sec CNT100;
   1:  PR[91,1] = PR[90,1] + 71.171;
   1:  PR[91,2] = PR[90,2] + -28.167;
   1:  PR[91,3] = PR[90,3] + 141.077;
   1:L PR[91] R[100]mm/sec CNT100;
   1:  PR[91,1] = PR[90,1] + 72.023;
   1:  PR[91,2] = PR[90,2] + -27.583;
   1:  PR[91,3] = PR[90,3] + 141.083;
   1:L PR[91] R[100]mm/sec CNT100;
   1:  PR[91,1] = PR[90,1] + 78.562;
   1:  PR[91,2] = PR[90,2] + -22.936;
   1:  PR[91,3] = PR[90,3] + 141.089;
   1:L PR[91] R[100]mm/sec CNT100;
   1:  PR[91,1] = PR[90,1] + 79.231;
   1:  PR[91,2] = PR[90,2] + -22.336;
   1:  PR[91,3] = PR[90,3] + 141.134;
   1:L PR[91] R[100]mm/sec CNT100;
   1:  PR[91,1] = PR[90,1] + 79.796;
   1:  PR[91,2] = PR[90,2] + -21.663;
   1:  PR[91,3] = PR[90,3] + 141.139;
   1:L PR[91] R[100]mm/sec CNT100;
   1:  PR[91,1] = PR[90,1] + 84.498;
   1:  PR[91,2] = PR[90,2] + -15.985;
   1:  PR[91,3] = PR[90,3] + 141.144;
   1:L PR[91] R[100]mm/sec CNT100;
   1:  PR[91,1] = PR[90,1] + 84.872;
   1:  PR[91,2] = PR[90,2] + -15.381;
   1:  PR[91,3] = PR[90,3] + 141.186;
   1:L PR[91] R[100]mm/sec CNT100;
   1:  PR[91,1] = PR[90,1] + 85.183;
   1:  PR[91,2] = PR[90,2] + -14.645;
   1:  PR[91,3] = PR[90,3] + 141.190;
   1:L PR[91] R[100]mm/sec CNT100;
   1:  PR[91,1] = PR[90,1] + 87.956;
   1:  PR[91,2] = PR[90,2] + -8.438;
   1:  PR[91,3] = PR[90,3] + 141.194;
   1:L PR[91] R[100]mm/sec CNT100;
   1:  PR[91,1] = PR[90,1] + 88.096;
   1:  PR[91,2] = PR[90,2] + -7.874;
   1:  PR[91,3] = PR[90,3] + 141.233;
   1:L PR[91] R[100]mm/sec CNT100;
   1:  PR[91,1] = PR[90,1] + 88.161;
   1:  PR[91,2] = PR[90,2] + -7.077;
   1:  PR[91,3] = PR[90,3] + 141.236;
   1:L PR[91] R[100]mm/sec CNT100;
   1:  PR[91,1] = PR[90,1] + 89.069;
   1:  PR[91,2] = PR[90,2] + -0.670;
   1:  PR[91,3] = PR[90,3] + 141.241;
   1:L PR[91] R[100]mm/sec CNT100;
   1:  PR[91,1] = PR[90,1] + 89.018;
   1:  PR[91,2] = PR[90,2] + -0.044;
   1:  PR[91,3] = PR[90,3] + 141.277;
   1:L PR[91] R[100]mm/sec CNT100;
   1:  PR[91,1] = PR[90,1] + 88.110;
   1:  PR[91,2] = PR[90,2] + 6.358;
   1:  PR[91,3] = PR[90,3] + 141.281;
   1:L PR[91] R[100]mm/sec CNT100;
   1:  PR[91,1] = PR[90,1] + 87.951;
   1:  PR[91,2] = PR[90,2] + 6.999;
   1:  PR[91,3] = PR[90,3] + 141.317;
   1:L PR[91] R[100]mm/sec CNT100;
   1:  PR[91,1] = PR[90,1] + 87.640;
   1:  PR[91,2] = PR[90,2] + 7.731;
   1:  PR[91,3] = PR[90,3] + 141.321;
   1:L PR[91] R[100]mm/sec CNT100;
   1:  PR[91,1] = PR[90,1] + 84.881;
   1:  PR[91,2] = PR[90,2] + 13.907;
   1:  PR[91,3] = PR[90,3] + 141.325;
   1:L PR[91] R[100]mm/sec CNT100;
   1:  PR[91,1] = PR[90,1] + 84.497;
   1:  PR[91,2] = PR[90,2] + 14.527;
   1:  PR[91,3] = PR[90,3] + 141.364;
   1:L PR[91] R[100]mm/sec CNT100;
   1:  PR[91,1] = PR[90,1] + 79.224;
   1:  PR[91,2] = PR[90,2] + 20.884;
   1:  PR[91,3] = PR[90,3] + 141.368;
   1:L PR[91] R[100]mm/sec CNT100;
   1:  PR[91,1] = PR[90,1] + 78.570;
   1:  PR[91,2] = PR[90,2] + 21.470;
   1:  PR[91,3] = PR[90,3] + 141.415;
   1:L PR[91] R[100]mm/sec CNT100;
   1:  PR[91,1] = PR[90,1] + 77.570;
   1:  PR[91,2] = PR[90,2] + 22.159;
   1:  PR[91,3] = PR[90,3] + 141.419;
   1:L PR[91] R[100]mm/sec CNT100;
   1:  PR[91,1] = PR[90,1] + 71.153;
   1:  PR[91,2] = PR[90,2] + 26.718;
   1:  PR[91,3] = PR[90,3] + 141.426;
   1:L PR[91] R[100]mm/sec CNT100;
   1:  PR[91,1] = PR[90,1] + 70.160;
   1:  PR[91,2] = PR[90,2] + 27.226;
   1:  PR[91,3] = PR[90,3] + 141.471;
   1:L PR[91] R[100]mm/sec CNT100;
   1:  PR[91,1] = PR[90,1] + 68.725;
   1:  PR[91,2] = PR[90,2] + 27.762;
   1:  PR[91,3] = PR[90,3] + 141.477;
   1:L PR[91] R[100]mm/sec CNT100;
   1:  PR[91,1] = PR[90,1] + 61.060;
   1:  PR[91,2] = PR[90,2] + 30.696;
   1:  PR[91,3] = PR[90,3] + 141.486;
   1:L PR[91] R[100]mm/sec CNT100;
   1:  PR[91,1] = PR[90,1] + 59.618;
   1:  PR[91,2] = PR[90,2] + 31.042;
   1:  PR[91,3] = PR[90,3] + 141.532;
   1:L PR[91] R[100]mm/sec CNT100;
   1:  PR[91,1] = PR[90,1] + 55.599;
   1:  PR[91,2] = PR[90,2] + 31.783;
   1:  PR[91,3] = PR[90,3] + 141.541;
   1:L PR[91] R[100]mm/sec CNT100;
   1:  PR[91,1] = PR[90,1] + 53.888;
   1:  PR[91,2] = PR[90,2] + 31.992;
   1:  PR[91,3] = PR[90,3] + 141.564;
   1:L PR[91] R[100]mm/sec CNT100;
   1:  PR[91,1] = PR[90,1] + 49.955;
   1:  PR[91,2] = PR[90,2] + 32.232;
   1:  PR[91,3] = PR[90,3] + 141.573;
   1:L PR[91] R[100]mm/sec CNT100;
   1:  PR[91,1] = PR[90,1] + 48.021;
   1:  PR[91,2] = PR[90,2] + 32.250;
   1:  PR[91,3] = PR[90,3] + 141.596;
   1:L PR[91] R[100]mm/sec CNT100;
   1:  PR[91,1] = PR[90,1] + 44.363;
   1:  PR[91,2] = PR[90,2] + 32.026;
   1:  PR[91,3] = PR[90,3] + 141.607;
   1:L PR[91] R[100]mm/sec CNT100;
   1:  PR[91,1] = PR[90,1] + 42.345;
   1:  PR[91,2] = PR[90,2] + 31.825;
   1:  PR[91,3] = PR[90,3] + 141.627;
   1:L PR[91] R[100]mm/sec CNT100;
   1:  PR[91,1] = PR[90,1] + 39.128;
   1:  PR[91,2] = PR[90,2] + 31.231;
   1:  PR[91,3] = PR[90,3] + 141.639;
   1:L PR[91] R[100]mm/sec CNT100;
   1:  PR[91,1] = PR[90,1] + 36.916;
   1:  PR[91,2] = PR[90,2] + 30.773;
   1:  PR[91,3] = PR[90,3] + 141.657;
   1:L PR[91] R[100]mm/sec CNT100;
   1:  PR[91,1] = PR[90,1] + 34.040;
   1:  PR[91,2] = PR[90,2] + 29.852;
   1:  PR[91,3] = PR[90,3] + 141.670;
   1:L PR[91] R[100]mm/sec CNT100;
   1:  PR[91,1] = PR[90,1] + 29.984;
   1:  PR[91,2] = PR[90,2] + 28.124;
   1:  PR[91,3] = PR[90,3] + 141.687;
   1:L PR[91] R[100]mm/sec CNT100;
   1:  PR[91,1] = PR[90,1] + 27.198;
   1:  PR[91,2] = PR[90,2] + 27.057;
   1:  PR[91,3] = PR[90,3] + 141.712;
   1:L PR[91] R[100]mm/sec CNT100;
   1:  PR[91,1] = PR[90,1] + 23.620;
   1:  PR[91,2] = PR[90,2] + 24.923;
   1:  PR[91,3] = PR[90,3] + 141.729;
   1:L PR[91] R[100]mm/sec CNT100;
   1:  PR[91,1] = PR[90,1] + 21.503;
   1:  PR[91,2] = PR[90,2] + 23.351;
   1:  PR[91,3] = PR[90,3] + 141.752;
   1:L PR[91] R[100]mm/sec CNT100;
   1:  PR[91,1] = PR[90,1] + 19.848;
   1:  PR[91,2] = PR[90,2] + 22.066;
   1:  PR[91,3] = PR[90,3] + 141.767;
   1:L PR[91] R[100]mm/sec CNT100;
   1:  PR[91,1] = PR[90,1] + 19.293;
   1:  PR[91,2] = PR[90,2] + 21.591;
   1:  PR[91,3] = PR[90,3] + 141.779;
   1:L PR[91] R[100]mm/sec CNT100;
   1:  PR[91,1] = PR[90,1] + 16.826;
   1:  PR[91,2] = PR[90,2] + 19.137;
   1:  PR[91,3] = PR[90,3] + 141.783;
   1:L PR[91] R[100]mm/sec CNT100;
   1:  PR[91,1] = PR[90,1] + 15.149;
   1:  PR[91,2] = PR[90,2] + 17.098;
   1:  PR[91,3] = PR[90,3] + 141.803;
   1:L PR[91] R[100]mm/sec CNT100;
   1:  PR[91,1] = PR[90,1] + 13.798;
   1:  PR[91,2] = PR[90,2] + 15.341;
   1:  PR[91,3] = PR[90,3] + 141.818;
   1:L PR[91] R[100]mm/sec CNT100;
   1:  PR[91,1] = PR[90,1] + 11.087;
   1:  PR[91,2] = PR[90,2] + 10.465;
   1:  PR[91,3] = PR[90,3] + 141.830;
   1:L PR[91] R[100]mm/sec CNT100;
   1:  PR[91,1] = PR[90,1] + 10.892;
   1:  PR[91,2] = PR[90,2] + 9.971;
   1:  PR[91,3] = PR[90,3] + 141.862;
   1:L PR[91] R[100]mm/sec CNT100;
   1:  PR[91,1] = PR[90,1] + 9.287;
   1:  PR[91,2] = PR[90,2] + 4.874;
   1:  PR[91,3] = PR[90,3] + 141.865;
   1:L PR[91] R[100]mm/sec CNT100;
   1:  PR[91] = PR[90];
   1:  PR[91,1] = PR[90,1] + 9.611;
   1:  PR[91,2] = PR[90,2] + -0.060;
   1:  PR[91,3] = PR[90,3] + 143.195;
   1:L PR[91] R[100]mm/sec CNT100;
   1:  PR[91,1] = PR[90,1] + 9.563;
   1:  PR[91,2] = PR[90,2] + -0.700;
   1:  PR[91,3] = PR[90,3] + 141.922;
   1:L PR[91] R[100]mm/sec CNT100;
   1:  PR[91,1] = PR[90,1] + 10.049;
   1:  PR[91,2] = PR[90,2] + -5.313;
   1:  PR[91,3] = PR[90,3] + 141.925;
   1:L PR[91] R[100]mm/sec CNT100;
   1:  PR[91,1] = PR[90,1] + 10.108;
   1:  PR[91,2] = PR[90,2] + -6.100;
   1:  PR[91,3] = PR[90,3] + 141.951;
   1:L PR[91] R[100]mm/sec CNT100;
   1:  PR[91,1] = PR[90,1] + 10.281;
   1:  PR[91,2] = PR[90,2] + -6.851;
   1:  PR[91,3] = PR[90,3] + 141.956;
   1:L PR[91] R[100]mm/sec CNT100;
   1:  PR[91,1] = PR[90,1] + 11.535;
   1:  PR[91,2] = PR[90,2] + -10.829;
   1:  PR[91,3] = PR[90,3] + 141.960;
   1:L PR[91] R[100]mm/sec CNT100;
   1:  PR[91,1] = PR[90,1] + 12.060;
   1:  PR[91,2] = PR[90,2] + -12.161;
   1:  PR[91,3] = PR[90,3] + 141.984;
   1:L PR[91] R[100]mm/sec CNT100;
   1:  PR[91,1] = PR[90,1] + 13.501;
   1:  PR[91,2] = PR[90,2] + -14.772;
   1:  PR[91,3] = PR[90,3] + 141.992;
   1:L PR[91] R[100]mm/sec CNT100;
   1:  PR[91,1] = PR[90,1] + 14.603;
   1:  PR[91,2] = PR[90,2] + -16.716;
   1:  PR[91,3] = PR[90,3] + 142.009;
   1:L PR[91] R[100]mm/sec CNT100;
   1:  PR[91,1] = PR[90,1] + 16.647;
   1:  PR[91,2] = PR[90,2] + -19.376;
   1:  PR[91,3] = PR[90,3] + 142.021;
   1:L PR[91] R[100]mm/sec CNT100;
   1:  PR[91,1] = PR[90,1] + 17.425;
   1:  PR[91,2] = PR[90,2] + -20.322;
   1:  PR[91,3] = PR[90,3] + 142.040;
   1:L PR[91] R[100]mm/sec CNT100;
   1:  PR[91,1] = PR[90,1] + 20.374;
   1:  PR[91,2] = PR[90,2] + -23.257;
   1:  PR[91,3] = PR[90,3] + 142.047;
   1:L PR[91] R[100]mm/sec CNT100;
   1:  PR[91,1] = PR[90,1] + 23.000;
   1:  PR[91,2] = PR[90,2] + -25.259;
   1:  PR[91,3] = PR[90,3] + 142.071;
   1:L PR[91] R[100]mm/sec CNT100;
   1:  PR[91,1] = PR[90,1] + 25.053;
   1:  PR[91,2] = PR[90,2] + -26.717;
   1:  PR[91,3] = PR[90,3] + 142.089;
   1:L PR[91] R[100]mm/sec CNT100;
   1:  PR[91,1] = PR[90,1] + 28.058;
   1:  PR[91,2] = PR[90,2] + -28.510;
   1:  PR[91,3] = PR[90,3] + 142.104;
   1:L PR[91] R[100]mm/sec CNT100;
   1:  PR[91,1] = PR[90,1] + 30.130;
   1:  PR[91,2] = PR[90,2] + -29.436;
   1:  PR[91,3] = PR[90,3] + 142.123;
   1:L PR[91] R[100]mm/sec CNT100;
   1:  PR[91,1] = PR[90,1] + 31.798;
   1:  PR[91,2] = PR[90,2] + -29.920;
   1:  PR[91,3] = PR[90,3] + 142.136;
   1:L PR[91] R[100]mm/sec CNT100;
   1:  PR[91,1] = PR[90,1] + 37.905;
   1:  PR[91,2] = PR[90,2] + -32.258;
   1:  PR[91,3] = PR[90,3] + 142.146;
   1:L PR[91] R[100]mm/sec CNT100;
   1:  PR[91,1] = PR[90,1] + 39.670;
   1:  PR[91,2] = PR[90,2] + -32.623;
   1:  PR[91,3] = PR[90,3] + 142.183;
   1:L PR[91] R[100]mm/sec CNT100;
   1:  PR[91,1] = PR[90,1] + 43.332;
   1:  PR[91,2] = PR[90,2] + -33.299;
   1:  PR[91,3] = PR[90,3] + 142.193;
   1:L PR[91] R[100]mm/sec CNT100;
   1:  PR[91,1] = PR[90,1] + 44.992;
   1:  PR[91,2] = PR[90,2] + -33.464;
   1:  PR[91,3] = PR[90,3] + 142.214;
   1:L PR[91] R[100]mm/sec CNT100;
   1:  PR[91,1] = PR[90,1] + 49.052;
   1:  PR[91,2] = PR[90,2] + -33.712;
   1:  PR[91,3] = PR[90,3] + 142.224;
   1:L PR[91] R[100]mm/sec CNT100;
   1:  PR[91,1] = PR[90,1] + 50.640;
   1:  PR[91,2] = PR[90,2] + -33.698;
   1:  PR[91,3] = PR[90,3] + 142.247;
   1:L PR[91] R[100]mm/sec CNT100;
   1:  PR[91,1] = PR[90,1] + 54.929;
   1:  PR[91,2] = PR[90,2] + -33.435;
   1:  PR[91,3] = PR[90,3] + 142.256;
   1:L PR[91] R[100]mm/sec CNT100;
   1:  PR[91,1] = PR[90,1] + 56.333;
   1:  PR[91,2] = PR[90,2] + -33.264;
   1:  PR[91,3] = PR[90,3] + 142.280;
   1:L PR[91] R[100]mm/sec CNT100;
   1:  PR[91,1] = PR[90,1] + 60.660;
   1:  PR[91,2] = PR[90,2] + -32.465;
   1:  PR[91,3] = PR[90,3] + 142.288;
   1:L PR[91] R[100]mm/sec CNT100;
   1:  PR[91,1] = PR[90,1] + 61.832;
   1:  PR[91,2] = PR[90,2] + -32.184;
   1:  PR[91,3] = PR[90,3] + 142.313;
   1:L PR[91] R[100]mm/sec CNT100;
   1:  PR[91,1] = PR[90,1] + 71.174;
   1:  PR[91,2] = PR[90,2] + -28.618;
   1:  PR[91,3] = PR[90,3] + 142.319;
   1:L PR[91] R[100]mm/sec CNT100;
   1:  PR[91,1] = PR[90,1] + 71.982;
   1:  PR[91,2] = PR[90,2] + -28.205;
   1:  PR[91,3] = PR[90,3] + 142.376;
   1:L PR[91] R[100]mm/sec CNT100;
   1:  PR[91,1] = PR[90,1] + 72.670;
   1:  PR[91,2] = PR[90,2] + -27.732;
   1:  PR[91,3] = PR[90,3] + 142.381;
   1:L PR[91] R[100]mm/sec CNT100;
   1:  PR[91,1] = PR[90,1] + 79.534;
   1:  PR[91,2] = PR[90,2] + -22.855;
   1:  PR[91,3] = PR[90,3] + 142.386;
   1:L PR[91] R[100]mm/sec CNT100;
   1:  PR[91,1] = PR[90,1] + 80.054;
   1:  PR[91,2] = PR[90,2] + -22.389;
   1:  PR[91,3] = PR[90,3] + 142.433;
   1:L PR[91] R[100]mm/sec CNT100;
   1:  PR[91,1] = PR[90,1] + 85.422;
   1:  PR[91,2] = PR[90,2] + -15.914;
   1:  PR[91,3] = PR[90,3] + 142.437;
   1:L PR[91] R[100]mm/sec CNT100;
   1:  PR[91,1] = PR[90,1] + 85.708;
   1:  PR[91,2] = PR[90,2] + -15.453;
   1:  PR[91,3] = PR[90,3] + 142.485;
   1:L PR[91] R[100]mm/sec CNT100;
   1:  PR[91,1] = PR[90,1] + 85.958;
   1:  PR[91,2] = PR[90,2] + -14.862;
   1:  PR[91,3] = PR[90,3] + 142.488;
   1:L PR[91] R[100]mm/sec CNT100;
   1:  PR[91,1] = PR[90,1] + 88.845;
   1:  PR[91,2] = PR[90,2] + -8.398;
   1:  PR[91,3] = PR[90,3] + 142.492;
   1:L PR[91] R[100]mm/sec CNT100;
   1:  PR[91,1] = PR[90,1] + 88.948;
   1:  PR[91,2] = PR[90,2] + -7.983;
   1:  PR[91,3] = PR[90,3] + 142.532;
   1:L PR[91] R[100]mm/sec CNT100;
   1:  PR[91,1] = PR[90,1] + 89.001;
   1:  PR[91,2] = PR[90,2] + -7.337;
   1:  PR[91,3] = PR[90,3] + 142.534;
   1:L PR[91] R[100]mm/sec CNT100;
   1:  PR[91,1] = PR[90,1] + 89.946;
   1:  PR[91,2] = PR[90,2] + -0.670;
   1:  PR[91,3] = PR[90,3] + 142.538;
   1:L PR[91] R[100]mm/sec CNT100;
   1:  PR[91,1] = PR[90,1] + 89.908;
   1:  PR[91,2] = PR[90,2] + -0.197;
   1:  PR[91,3] = PR[90,3] + 142.576;
   1:L PR[91] R[100]mm/sec CNT100;
   1:  PR[91,1] = PR[90,1] + 88.962;
   1:  PR[91,2] = PR[90,2] + 6.467;
   1:  PR[91,3] = PR[90,3] + 142.578;
   1:L PR[91] R[100]mm/sec CNT100;
   1:  PR[91,1] = PR[90,1] + 88.840;
   1:  PR[91,2] = PR[90,2] + 6.958;
   1:  PR[91,3] = PR[90,3] + 142.616;
   1:L PR[91] R[100]mm/sec CNT100;
   1:  PR[91,1] = PR[90,1] + 88.594;
   1:  PR[91,2] = PR[90,2] + 7.540;
   1:  PR[91,3] = PR[90,3] + 142.619;
   1:L PR[91] R[100]mm/sec CNT100;
   1:  PR[91,1] = PR[90,1] + 85.717;
   1:  PR[91,2] = PR[90,2] + 13.980;
   1:  PR[91,3] = PR[90,3] + 142.623;
   1:L PR[91] R[100]mm/sec CNT100;
   1:  PR[91,1] = PR[90,1] + 85.421;
   1:  PR[91,2] = PR[90,2] + 14.457;
   1:  PR[91,3] = PR[90,3] + 142.663;
   1:L PR[91] R[100]mm/sec CNT100;
   1:  PR[91,1] = PR[90,1] + 80.051;
   1:  PR[91,2] = PR[90,2] + 20.933;
   1:  PR[91,3] = PR[90,3] + 142.666;
   1:L PR[91] R[100]mm/sec CNT100;
   1:  PR[91,1] = PR[90,1] + 79.541;
   1:  PR[91,2] = PR[90,2] + 21.390;
   1:  PR[91,3] = PR[90,3] + 142.713;
   1:L PR[91] R[100]mm/sec CNT100;
   1:  PR[91,1] = PR[90,1] + 78.725;
   1:  PR[91,2] = PR[90,2] + 21.953;
   1:  PR[91,3] = PR[90,3] + 142.717;
   1:L PR[91] R[100]mm/sec CNT100;
   1:  PR[91,1] = PR[90,1] + 71.963;
   1:  PR[91,2] = PR[90,2] + 26.756;
   1:  PR[91,3] = PR[90,3] + 142.723;
   1:L PR[91] R[100]mm/sec CNT100;
   1:  PR[91,1] = PR[90,1] + 71.170;
   1:  PR[91,2] = PR[90,2] + 27.161;
   1:  PR[91,3] = PR[90,3] + 142.770;
   1:L PR[91] R[100]mm/sec CNT100;
   1:  PR[91,1] = PR[90,1] + 61.828;
   1:  PR[91,2] = PR[90,2] + 30.727;
   1:  PR[91,3] = PR[90,3] + 142.775;
   1:L PR[91] R[100]mm/sec CNT100;
   1:  PR[91,1] = PR[90,1] + 60.656;
   1:  PR[91,2] = PR[90,2] + 31.007;
   1:  PR[91,3] = PR[90,3] + 142.831;
   1:L PR[91] R[100]mm/sec CNT100;
   1:  PR[91,1] = PR[90,1] + 56.329;
   1:  PR[91,2] = PR[90,2] + 31.806;
   1:  PR[91,3] = PR[90,3] + 142.838;
   1:L PR[91] R[100]mm/sec CNT100;
   1:  PR[91,1] = PR[90,1] + 54.925;
   1:  PR[91,2] = PR[90,2] + 31.977;
   1:  PR[91,3] = PR[90,3] + 142.863;
   1:L PR[91] R[100]mm/sec CNT100;
   1:  PR[91,1] = PR[90,1] + 50.636;
   1:  PR[91,2] = PR[90,2] + 32.239;
   1:  PR[91,3] = PR[90,3] + 142.871;
   1:L PR[91] R[100]mm/sec CNT100;
   1:  PR[91,1] = PR[90,1] + 49.048;
   1:  PR[91,2] = PR[90,2] + 32.253;
   1:  PR[91,3] = PR[90,3] + 142.895;
   1:L PR[91] R[100]mm/sec CNT100;
   1:  PR[91,1] = PR[90,1] + 44.987;
   1:  PR[91,2] = PR[90,2] + 32.004;
   1:  PR[91,3] = PR[90,3] + 142.904;
   1:L PR[91] R[100]mm/sec CNT100;
   1:  PR[91,1] = PR[90,1] + 43.328;
   1:  PR[91,2] = PR[90,2] + 31.840;
   1:  PR[91,3] = PR[90,3] + 142.927;
   1:L PR[91] R[100]mm/sec CNT100;
   1:  PR[91,1] = PR[90,1] + 39.666;
   1:  PR[91,2] = PR[90,2] + 31.164;
   1:  PR[91,3] = PR[90,3] + 142.937;
   1:L PR[91] R[100]mm/sec CNT100;
   1:  PR[91,1] = PR[90,1] + 37.846;
   1:  PR[91,2] = PR[90,2] + 30.787;
   1:  PR[91,3] = PR[90,3] + 142.958;
   1:L PR[91] R[100]mm/sec CNT100;
   1:  PR[91,1] = PR[90,1] + 35.485;
   1:  PR[91,2] = PR[90,2] + 30.030;
   1:  PR[91,3] = PR[90,3] + 142.968;
   1:L PR[91] R[100]mm/sec CNT100;
   1:  PR[91,1] = PR[90,1] + 32.117;
   1:  PR[91,2] = PR[90,2] + 28.595;
   1:  PR[91,3] = PR[90,3] + 142.982;
   1:L PR[91] R[100]mm/sec CNT100;
   1:  PR[91,1] = PR[90,1] + 28.008;
   1:  PR[91,2] = PR[90,2] + 27.022;
   1:  PR[91,3] = PR[90,3] + 143.003;
   1:L PR[91] R[100]mm/sec CNT100;
   1:  PR[91,1] = PR[90,1] + 25.070;
   1:  PR[91,2] = PR[90,2] + 25.269;
   1:  PR[91,3] = PR[90,3] + 143.028;
   1:L PR[91] R[100]mm/sec CNT100;
   1:  PR[91,1] = PR[90,1] + 20.662;
   1:  PR[91,2] = PR[90,2] + 21.997;
   1:  PR[91,3] = PR[90,3] + 143.047;
   1:L PR[91] R[100]mm/sec CNT100;
   1:  PR[91,1] = PR[90,1] + 20.350;
   1:  PR[91,2] = PR[90,2] + 21.775;
   1:  PR[91,3] = PR[90,3] + 143.078;
   1:L PR[91] R[100]mm/sec CNT100;
   1:  PR[91,1] = PR[90,1] + 17.426;
   1:  PR[91,2] = PR[90,2] + 18.864;
   1:  PR[91,3] = PR[90,3] + 143.080;
   1:L PR[91] R[100]mm/sec CNT100;
   1:  PR[91,1] = PR[90,1] + 16.648;
   1:  PR[91,2] = PR[90,2] + 17.919;
   1:  PR[91,3] = PR[90,3] + 143.103;
   1:L PR[91] R[100]mm/sec CNT100;
   1:  PR[91,1] = PR[90,1] + 14.607;
   1:  PR[91,2] = PR[90,2] + 15.264;
   1:  PR[91,3] = PR[90,3] + 143.110;
   1:L PR[91] R[100]mm/sec CNT100;
   1:  PR[91,1] = PR[90,1] + 12.059;
   1:  PR[91,2] = PR[90,2] + 10.699;
   1:  PR[91,3] = PR[90,3] + 143.129;
   1:L PR[91] R[100]mm/sec CNT100;
   1:  PR[91,1] = PR[90,1] + 11.536;
   1:  PR[91,2] = PR[90,2] + 9.372;
   1:  PR[91,3] = PR[90,3] + 143.159;
   1:L PR[91] R[100]mm/sec CNT100;
   1:  PR[91,1] = PR[90,1] + 10.282;
   1:  PR[91,2] = PR[90,2] + 5.393;
   1:  PR[91,3] = PR[90,3] + 143.167;
   1:L PR[91] R[100]mm/sec CNT100;
   1:  PR[91,1] = PR[90,1] + 10.101;
   1:  PR[91,2] = PR[90,2] + 4.613;
   1:  PR[91,3] = PR[90,3] + 143.190;
   1:L PR[91] R[100]mm/sec CNT100;
   1:  PR[91] = PR[90];
   1:  PR[91,1] = PR[90,1] + 10.551;
   1:  PR[91,2] = PR[90,2] + 0.887;
   1:  PR[91,3] = PR[90,3] + 144.495;
   1:L PR[91] R[100]mm/sec CNT100;
   1:  PR[91,1] = PR[90,1] + 10.431;
   1:  PR[91,2] = PR[90,2] + -0.700;
   1:  PR[91,3] = PR[90,3] + 143.214;
   1:L PR[91] R[100]mm/sec CNT100;
   1:  PR[91,1] = PR[90,1] + 10.787;
   1:  PR[91,2] = PR[90,2] + -4.081;
   1:  PR[91,3] = PR[90,3] + 143.223;
   1:L PR[91] R[100]mm/sec CNT100;
   1:  PR[91,1] = PR[90,1] + 10.913;
   1:  PR[91,2] = PR[90,2] + -5.760;
   1:  PR[91,3] = PR[90,3] + 143.242;
   1:L PR[91] R[100]mm/sec CNT100;
   1:  PR[91,1] = PR[90,1] + 11.309;
   1:  PR[91,2] = PR[90,2] + -7.468;
   1:  PR[91,3] = PR[90,3] + 143.252;
   1:L PR[91] R[100]mm/sec CNT100;
   1:  PR[91,1] = PR[90,1] + 12.179;
   1:  PR[91,2] = PR[90,2] + -10.231;
   1:  PR[91,3] = PR[90,3] + 143.262;
   1:L PR[91] R[100]mm/sec CNT100;
   1:  PR[91,1] = PR[90,1] + 13.033;
   1:  PR[91,2] = PR[90,2] + -12.397;
   1:  PR[91,3] = PR[90,3] + 143.278;
   1:L PR[91] R[100]mm/sec CNT100;
   1:  PR[91,1] = PR[90,1] + 13.936;
   1:  PR[91,2] = PR[90,2] + -14.032;
   1:  PR[91,3] = PR[90,3] + 143.291;
   1:L PR[91] R[100]mm/sec CNT100;
   1:  PR[91,1] = PR[90,1] + 15.413;
   1:  PR[91,2] = PR[90,2] + -16.640;
   1:  PR[91,3] = PR[90,3] + 143.302;
   1:L PR[91] R[100]mm/sec CNT100;
   1:  PR[91,1] = PR[90,1] + 18.088;
   1:  PR[91,2] = PR[90,2] + -20.112;
   1:  PR[91,3] = PR[90,3] + 143.319;
   1:L PR[91] R[100]mm/sec CNT100;
   1:  PR[91,1] = PR[90,1] + 21.086;
   1:  PR[91,2] = PR[90,2] + -23.109;
   1:  PR[91,3] = PR[90,3] + 143.344;
   1:L PR[91] R[100]mm/sec CNT100;
   1:  PR[91,1] = PR[90,1] + 23.155;
   1:  PR[91,2] = PR[90,2] + -24.686;
   1:  PR[91,3] = PR[90,3] + 143.368;
   1:L PR[91] R[100]mm/sec CNT100;
   1:  PR[91,1] = PR[90,1] + 26.503;
   1:  PR[91,2] = PR[90,2] + -27.064;
   1:  PR[91,3] = PR[90,3] + 143.382;
   1:L PR[91] R[100]mm/sec CNT100;
   1:  PR[91,1] = PR[90,1] + 28.869;
   1:  PR[91,2] = PR[90,2] + -28.475;
   1:  PR[91,3] = PR[90,3] + 143.405;
   1:L PR[91] R[100]mm/sec CNT100;
   1:  PR[91,1] = PR[90,1] + 30.477;
   1:  PR[91,2] = PR[90,2] + -29.194;
   1:  PR[91,3] = PR[90,3] + 143.421;
   1:L PR[91] R[100]mm/sec CNT100;
   1:  PR[91,1] = PR[90,1] + 31.798;
   1:  PR[91,2] = PR[90,2] + -29.577;
   1:  PR[91,3] = PR[90,3] + 143.431;
   1:L PR[91] R[100]mm/sec CNT100;
   1:  PR[91,1] = PR[90,1] + 38.836;
   1:  PR[91,2] = PR[90,2] + -32.271;
   1:  PR[91,3] = PR[90,3] + 143.439;
   1:L PR[91] R[100]mm/sec CNT100;
   1:  PR[91,1] = PR[90,1] + 40.209;
   1:  PR[91,2] = PR[90,2] + -32.556;
   1:  PR[91,3] = PR[90,3] + 143.481;
   1:L PR[91] R[100]mm/sec CNT100;
   1:  PR[91,1] = PR[90,1] + 44.315;
   1:  PR[91,2] = PR[90,2] + -33.313;
   1:  PR[91,3] = PR[90,3] + 143.489;
   1:L PR[91] R[100]mm/sec CNT100;
   1:  PR[91,1] = PR[90,1] + 45.616;
   1:  PR[91,2] = PR[90,2] + -33.443;
   1:  PR[91,3] = PR[90,3] + 143.513;
   1:L PR[91] R[100]mm/sec CNT100;
   1:  PR[91,1] = PR[90,1] + 50.078;
   1:  PR[91,2] = PR[90,2] + -33.715;
   1:  PR[91,3] = PR[90,3] + 143.520;
   1:L PR[91] R[100]mm/sec CNT100;
   1:  PR[91,1] = PR[90,1] + 51.322;
   1:  PR[91,2] = PR[90,2] + -33.704;
   1:  PR[91,3] = PR[90,3] + 143.546;
   1:L PR[91] R[100]mm/sec CNT100;
   1:  PR[91,1] = PR[90,1] + 55.966;
   1:  PR[91,2] = PR[90,2] + -33.420;
   1:  PR[91,3] = PR[90,3] + 143.553;
   1:L PR[91] R[100]mm/sec CNT100;
   1:  PR[91,1] = PR[90,1] + 57.063;
   1:  PR[91,2] = PR[90,2] + -33.286;
   1:  PR[91,3] = PR[90,3] + 143.579;
   1:L PR[91] R[100]mm/sec CNT100;
   1:  PR[91,1] = PR[90,1] + 61.699;
   1:  PR[91,2] = PR[90,2] + -32.430;
   1:  PR[91,3] = PR[90,3] + 143.585;
   1:L PR[91] R[100]mm/sec CNT100;
   1:  PR[91,1] = PR[90,1] + 62.598;
   1:  PR[91,2] = PR[90,2] + -32.215;
   1:  PR[91,3] = PR[90,3] + 143.612;
   1:L PR[91] R[100]mm/sec CNT100;
   1:  PR[91,1] = PR[90,1] + 72.189;
   1:  PR[91,2] = PR[90,2] + -28.551;
   1:  PR[91,3] = PR[90,3] + 143.617;
   1:L PR[91] R[100]mm/sec CNT100;
   1:  PR[91,1] = PR[90,1] + 72.792;
   1:  PR[91,2] = PR[90,2] + -28.242;
   1:  PR[91,3] = PR[90,3] + 143.675;
   1:L PR[91] R[100]mm/sec CNT100;
   1:  PR[91,1] = PR[90,1] + 73.318;
   1:  PR[91,2] = PR[90,2] + -27.881;
   1:  PR[91,3] = PR[90,3] + 143.679;
   1:L PR[91] R[100]mm/sec CNT100;
   1:  PR[91,1] = PR[90,1] + 80.505;
   1:  PR[91,2] = PR[90,2] + -22.775;
   1:  PR[91,3] = PR[90,3] + 143.682;
   1:L PR[91] R[100]mm/sec CNT100;
   1:  PR[91,1] = PR[90,1] + 80.881;
   1:  PR[91,2] = PR[90,2] + -22.437;
   1:  PR[91,3] = PR[90,3] + 143.732;
   1:L PR[91] R[100]mm/sec CNT100;
   1:  PR[91,1] = PR[90,1] + 86.346;
   1:  PR[91,2] = PR[90,2] + -15.844;
   1:  PR[91,3] = PR[90,3] + 143.735;
   1:L PR[91] R[100]mm/sec CNT100;
   1:  PR[91,1] = PR[90,1] + 86.543;
   1:  PR[91,2] = PR[90,2] + -15.526;
   1:  PR[91,3] = PR[90,3] + 143.783;
   1:L PR[91] R[100]mm/sec CNT100;
   1:  PR[91,1] = PR[90,1] + 86.733;
   1:  PR[91,2] = PR[90,2] + -15.079;
   1:  PR[91,3] = PR[90,3] + 143.786;
   1:L PR[91] R[100]mm/sec CNT100;
   1:  PR[91,1] = PR[90,1] + 89.735;
   1:  PR[91,2] = PR[90,2] + -8.357;
   1:  PR[91,3] = PR[90,3] + 143.788;
   1:L PR[91] R[100]mm/sec CNT100;
   1:  PR[91,1] = PR[90,1] + 89.800;
   1:  PR[91,2] = PR[90,2] + -8.093;
   1:  PR[91,3] = PR[90,3] + 143.830;
   1:L PR[91] R[100]mm/sec CNT100;
   1:  PR[91,1] = PR[90,1] + 89.841;
   1:  PR[91,2] = PR[90,2] + -7.597;
   1:  PR[91,3] = PR[90,3] + 143.831;
   1:L PR[91] R[100]mm/sec CNT100;
   1:  PR[91,1] = PR[90,1] + 90.823;
   1:  PR[91,2] = PR[90,2] + -0.670;
   1:  PR[91,3] = PR[90,3] + 143.834;
   1:L PR[91] R[100]mm/sec CNT100;
   1:  PR[91,1] = PR[90,1] + 90.797;
   1:  PR[91,2] = PR[90,2] + -0.348;
   1:  PR[91,3] = PR[90,3] + 143.874;
   1:L PR[91] R[100]mm/sec CNT100;
   1:  PR[91,1] = PR[90,1] + 89.815;
   1:  PR[91,2] = PR[90,2] + 6.577;
   1:  PR[91,3] = PR[90,3] + 143.876;
   1:L PR[91] R[100]mm/sec CNT100;
   1:  PR[91,1] = PR[90,1] + 89.730;
   1:  PR[91,2] = PR[90,2] + 6.918;
   1:  PR[91,3] = PR[90,3] + 143.915;
   1:L PR[91] R[100]mm/sec CNT100;
   1:  PR[91,1] = PR[90,1] + 89.547;
   1:  PR[91,2] = PR[90,2] + 7.350;
   1:  PR[91,3] = PR[90,3] + 143.917;
   1:L PR[91] R[100]mm/sec CNT100;
   1:  PR[91,1] = PR[90,1] + 86.552;
   1:  PR[91,2] = PR[90,2] + 14.053;
   1:  PR[91,3] = PR[90,3] + 143.920;
   1:L PR[91] R[100]mm/sec CNT100;
   1:  PR[91,1] = PR[90,1] + 86.345;
   1:  PR[91,2] = PR[90,2] + 14.387;
   1:  PR[91,3] = PR[90,3] + 143.961;
   1:L PR[91] R[100]mm/sec CNT100;
   1:  PR[91,1] = PR[90,1] + 80.878;
   1:  PR[91,2] = PR[90,2] + 20.981;
   1:  PR[91,3] = PR[90,3] + 143.963;
   1:L PR[91] R[100]mm/sec CNT100;
   1:  PR[91,1] = PR[90,1] + 80.512;
   1:  PR[91,2] = PR[90,2] + 21.309;
   1:  PR[91,3] = PR[90,3] + 144.012;
   1:L PR[91] R[100]mm/sec CNT100;
   1:  PR[91,1] = PR[90,1] + 79.879;
   1:  PR[91,2] = PR[90,2] + 21.746;
   1:  PR[91,3] = PR[90,3] + 144.015;
   1:L PR[91] R[100]mm/sec CNT100;
   1:  PR[91,1] = PR[90,1] + 72.773;
   1:  PR[91,2] = PR[90,2] + 26.793;
   1:  PR[91,3] = PR[90,3] + 144.019;
   1:L PR[91] R[100]mm/sec CNT100;
   1:  PR[91,1] = PR[90,1] + 72.185;
   1:  PR[91,2] = PR[90,2] + 27.094;
   1:  PR[91,3] = PR[90,3] + 144.068;
   1:L PR[91] R[100]mm/sec CNT100;
   1:  PR[91,1] = PR[90,1] + 62.594;
   1:  PR[91,2] = PR[90,2] + 30.757;
   1:  PR[91,3] = PR[90,3] + 144.072;
   1:L PR[91] R[100]mm/sec CNT100;
   1:  PR[91,1] = PR[90,1] + 61.694;
   1:  PR[91,2] = PR[90,2] + 30.973;
   1:  PR[91,3] = PR[90,3] + 144.130;
   1:L PR[91] R[100]mm/sec CNT100;
   1:  PR[91,1] = PR[90,1] + 57.058;
   1:  PR[91,2] = PR[90,2] + 31.828;
   1:  PR[91,3] = PR[90,3] + 144.135;
   1:L PR[91] R[100]mm/sec CNT100;
   1:  PR[91,1] = PR[90,1] + 55.962;
   1:  PR[91,2] = PR[90,2] + 31.961;
   1:  PR[91,3] = PR[90,3] + 144.162;
   1:L PR[91] R[100]mm/sec CNT100;
   1:  PR[91,1] = PR[90,1] + 51.318;
   1:  PR[91,2] = PR[90,2] + 32.245;
   1:  PR[91,3] = PR[90,3] + 144.168;
   1:L PR[91] R[100]mm/sec CNT100;
   1:  PR[91,1] = PR[90,1] + 50.074;
   1:  PR[91,2] = PR[90,2] + 32.257;
   1:  PR[91,3] = PR[90,3] + 144.194;
   1:L PR[91] R[100]mm/sec CNT100;
   1:  PR[91,1] = PR[90,1] + 45.612;
   1:  PR[91,2] = PR[90,2] + 31.983;
   1:  PR[91,3] = PR[90,3] + 144.201;
   1:L PR[91] R[100]mm/sec CNT100;
   1:  PR[91,1] = PR[90,1] + 44.311;
   1:  PR[91,2] = PR[90,2] + 31.854;
   1:  PR[91,3] = PR[90,3] + 144.227;
   1:L PR[91] R[100]mm/sec CNT100;
   1:  PR[91,1] = PR[90,1] + 40.205;
   1:  PR[91,2] = PR[90,2] + 31.096;
   1:  PR[91,3] = PR[90,3] + 144.234;
   1:L PR[91] R[100]mm/sec CNT100;
   1:  PR[91,1] = PR[90,1] + 38.777;
   1:  PR[91,2] = PR[90,2] + 30.800;
   1:  PR[91,3] = PR[90,3] + 144.258;
   1:L PR[91] R[100]mm/sec CNT100;
   1:  PR[91,1] = PR[90,1] + 36.929;
   1:  PR[91,2] = PR[90,2] + 30.208;
   1:  PR[91,3] = PR[90,3] + 144.266;
   1:L PR[91] R[100]mm/sec CNT100;
   1:  PR[91,1] = PR[90,1] + 34.250;
   1:  PR[91,2] = PR[90,2] + 29.067;
   1:  PR[91,3] = PR[90,3] + 144.277;
   1:L PR[91] R[100]mm/sec CNT100;
   1:  PR[91,1] = PR[90,1] + 28.819;
   1:  PR[91,2] = PR[90,2] + 26.987;
   1:  PR[91,3] = PR[90,3] + 144.293;
   1:L PR[91] R[100]mm/sec CNT100;
   1:  PR[91,1] = PR[90,1] + 26.519;
   1:  PR[91,2] = PR[90,2] + 25.615;
   1:  PR[91,3] = PR[90,3] + 144.326;
   1:L PR[91] R[100]mm/sec CNT100;
   1:  PR[91,1] = PR[90,1] + 23.012;
   1:  PR[91,2] = PR[90,2] + 23.011;
   1:  PR[91,3] = PR[90,3] + 144.341;
   1:L PR[91] R[100]mm/sec CNT100;
   1:  PR[91,1] = PR[90,1] + 21.062;
   1:  PR[91,2] = PR[90,2] + 21.625;
   1:  PR[91,3] = PR[90,3] + 144.366;
   1:L PR[91] R[100]mm/sec CNT100;
   1:  PR[91,1] = PR[90,1] + 18.088;
   1:  PR[91,2] = PR[90,2] + 18.654;
   1:  PR[91,3] = PR[90,3] + 144.379;
   1:L PR[91] R[100]mm/sec CNT100;
   1:  PR[91,1] = PR[90,1] + 15.416;
   1:  PR[91,2] = PR[90,2] + 15.186;
   1:  PR[91,3] = PR[90,3] + 144.403;
   1:L PR[91] R[100]mm/sec CNT100;
   1:  PR[91,1] = PR[90,1] + 13.031;
   1:  PR[91,2] = PR[90,2] + 10.933;
   1:  PR[91,3] = PR[90,3] + 144.428;
   1:L PR[91] R[100]mm/sec CNT100;
   1:  PR[91,1] = PR[90,1] + 12.180;
   1:  PR[91,2] = PR[90,2] + 8.773;
   1:  PR[91,3] = PR[90,3] + 144.455;
   1:L PR[91] R[100]mm/sec CNT100;
   1:  PR[91,1] = PR[90,1] + 11.309;
   1:  PR[91,2] = PR[90,2] + 6.009;
   1:  PR[91,3] = PR[90,3] + 144.469;
   1:L PR[91] R[100]mm/sec CNT100;
   1:  PR[91,1] = PR[90,1] + 10.906;
   1:  PR[91,2] = PR[90,2] + 4.272;
   1:  PR[91,3] = PR[90,3] + 144.485;
   1:L PR[91] R[100]mm/sec CNT100;
   1:  PR[91] = PR[90];
   1:  PR[91,1] = PR[90,1] + 11.492;
   1:  PR[91,2] = PR[90,2] + 1.834;
   1:  PR[91,3] = PR[90,3] + 145.795;
   1:L PR[91] R[100]mm/sec CNT100;
   1:  PR[91,1] = PR[90,1] + 11.300;
   1:  PR[91,2] = PR[90,2] + -0.700;
   1:  PR[91,3] = PR[90,3] + 144.507;
   1:L PR[91] R[100]mm/sec CNT100;
   1:  PR[91,1] = PR[90,1] + 11.526;
   1:  PR[91,2] = PR[90,2] + -2.849;
   1:  PR[91,3] = PR[90,3] + 144.521;
   1:L PR[91] R[100]mm/sec CNT100;
   1:  PR[91,1] = PR[90,1] + 11.719;
   1:  PR[91,2] = PR[90,2] + -5.420;
   1:  PR[91,3] = PR[90,3] + 144.533;
   1:L PR[91] R[100]mm/sec CNT100;
   1:  PR[91,1] = PR[90,1] + 12.336;
   1:  PR[91,2] = PR[90,2] + -8.084;
   1:  PR[91,3] = PR[90,3] + 144.548;
   1:L PR[91] R[100]mm/sec CNT100;
   1:  PR[91,1] = PR[90,1] + 12.823;
   1:  PR[91,2] = PR[90,2] + -9.632;
   1:  PR[91,3] = PR[90,3] + 144.564;
   1:L PR[91] R[100]mm/sec CNT100;
   1:  PR[91,1] = PR[90,1] + 14.003;
   1:  PR[91,2] = PR[90,2] + -12.625;
   1:  PR[91,3] = PR[90,3] + 144.573;
   1:L PR[91] R[100]mm/sec CNT100;
   1:  PR[91,1] = PR[90,1] + 16.219;
   1:  PR[91,2] = PR[90,2] + -16.556;
   1:  PR[91,3] = PR[90,3] + 144.591;
   1:L PR[91] R[100]mm/sec CNT100;
   1:  PR[91,1] = PR[90,1] + 18.085;
   1:  PR[91,2] = PR[90,2] + -18.939;
   1:  PR[91,3] = PR[90,3] + 144.616;
   1:L PR[91] R[100]mm/sec CNT100;
   1:  PR[91,1] = PR[90,1] + 19.576;
   1:  PR[91,2] = PR[90,2] + -20.740;
   1:  PR[91,3] = PR[90,3] + 144.633;
   1:L PR[91] R[100]mm/sec CNT100;
   1:  PR[91,1] = PR[90,1] + 21.797;
   1:  PR[91,2] = PR[90,2] + -22.959;
   1:  PR[91,3] = PR[90,3] + 144.647;
   1:L PR[91] R[100]mm/sec CNT100;
   1:  PR[91,1] = PR[90,1] + 23.310;
   1:  PR[91,2] = PR[90,2] + -24.113;
   1:  PR[91,3] = PR[90,3] + 144.664;
   1:L PR[91] R[100]mm/sec CNT100;
   1:  PR[91,1] = PR[90,1] + 27.954;
   1:  PR[91,2] = PR[90,2] + -27.411;
   1:  PR[91,3] = PR[90,3] + 144.675;
   1:L PR[91] R[100]mm/sec CNT100;
   1:  PR[91,1] = PR[90,1] + 29.680;
   1:  PR[91,2] = PR[90,2] + -28.441;
   1:  PR[91,3] = PR[90,3] + 144.707;
   1:L PR[91] R[100]mm/sec CNT100;
   1:  PR[91,1] = PR[90,1] + 30.824;
   1:  PR[91,2] = PR[90,2] + -28.952;
   1:  PR[91,3] = PR[90,3] + 144.719;
   1:L PR[91] R[100]mm/sec CNT100;
   1:  PR[91,1] = PR[90,1] + 31.799;
   1:  PR[91,2] = PR[90,2] + -29.235;
   1:  PR[91,3] = PR[90,3] + 144.726;
   1:L PR[91] R[100]mm/sec CNT100;
   1:  PR[91,1] = PR[90,1] + 39.767;
   1:  PR[91,2] = PR[90,2] + -32.285;
   1:  PR[91,3] = PR[90,3] + 144.732;
   1:L PR[91] R[100]mm/sec CNT100;
   1:  PR[91,1] = PR[90,1] + 40.749;
   1:  PR[91,2] = PR[90,2] + -32.488;
   1:  PR[91,3] = PR[90,3] + 144.780;
   1:L PR[91] R[100]mm/sec CNT100;
   1:  PR[91,1] = PR[90,1] + 45.298;
   1:  PR[91,2] = PR[90,2] + -33.328;
   1:  PR[91,3] = PR[90,3] + 144.785;
   1:L PR[91] R[100]mm/sec CNT100;
   1:  PR[91,1] = PR[90,1] + 46.241;
   1:  PR[91,2] = PR[90,2] + -33.421;
   1:  PR[91,3] = PR[90,3] + 144.812;
   1:L PR[91] R[100]mm/sec CNT100;
   1:  PR[91,1] = PR[90,1] + 51.105;
   1:  PR[91,2] = PR[90,2] + -33.719;
   1:  PR[91,3] = PR[90,3] + 144.817;
   1:L PR[91] R[100]mm/sec CNT100;
   1:  PR[91,1] = PR[90,1] + 52.004;
   1:  PR[91,2] = PR[90,2] + -33.711;
   1:  PR[91,3] = PR[90,3] + 144.844;
   1:L PR[91] R[100]mm/sec CNT100;
   1:  PR[91,1] = PR[90,1] + 57.003;
   1:  PR[91,2] = PR[90,2] + -33.404;
   1:  PR[91,3] = PR[90,3] + 144.849;
   1:L PR[91] R[100]mm/sec CNT100;
   1:  PR[91,1] = PR[90,1] + 57.793;
   1:  PR[91,2] = PR[90,2] + -33.308;
   1:  PR[91,3] = PR[90,3] + 144.878;
   1:L PR[91] R[100]mm/sec CNT100;
   1:  PR[91,1] = PR[90,1] + 62.737;
   1:  PR[91,2] = PR[90,2] + -32.395;
   1:  PR[91,3] = PR[90,3] + 144.882;
   1:L PR[91] R[100]mm/sec CNT100;
   1:  PR[91,1] = PR[90,1] + 63.373;
   1:  PR[91,2] = PR[90,2] + -32.243;
   1:  PR[91,3] = PR[90,3] + 144.911;
   1:L PR[91] R[100]mm/sec CNT100;
   1:  PR[91,1] = PR[90,1] + 63.893;
   1:  PR[91,2] = PR[90,2] + -32.050;
   1:  PR[91,3] = PR[90,3] + 144.914;
   1:L PR[91] R[100]mm/sec CNT100;
   1:  PR[91,1] = PR[90,1] + 73.204;
   1:  PR[91,2] = PR[90,2] + -28.484;
   1:  PR[91,3] = PR[90,3] + 144.918;
   1:L PR[91] R[100]mm/sec CNT100;
   1:  PR[91,1] = PR[90,1] + 73.589;
   1:  PR[91,2] = PR[90,2] + -28.287;
   1:  PR[91,3] = PR[90,3] + 144.974;
   1:L PR[91] R[100]mm/sec CNT100;
   1:  PR[91,1] = PR[90,1] + 81.477;
   1:  PR[91,2] = PR[90,2] + -22.693;
   1:  PR[91,3] = PR[90,3] + 144.976;
   1:L PR[91] R[100]mm/sec CNT100;
   1:  PR[91,1] = PR[90,1] + 81.708;
   1:  PR[91,2] = PR[90,2] + -22.486;
   1:  PR[91,3] = PR[90,3] + 145.031;
   1:L PR[91] R[100]mm/sec CNT100;
   1:  PR[91,1] = PR[90,1] + 87.270;
   1:  PR[91,2] = PR[90,2] + -15.774;
   1:  PR[91,3] = PR[90,3] + 145.033;
   1:L PR[91] R[100]mm/sec CNT100;
   1:  PR[91,1] = PR[90,1] + 87.389;
   1:  PR[91,2] = PR[90,2] + -15.582;
   1:  PR[91,3] = PR[90,3] + 145.082;
   1:L PR[91] R[100]mm/sec CNT100;
   1:  PR[91,1] = PR[90,1] + 90.624;
   1:  PR[91,2] = PR[90,2] + -8.318;
   1:  PR[91,3] = PR[90,3] + 145.083;
   1:L PR[91] R[100]mm/sec CNT100;
   1:  PR[91,1] = PR[90,1] + 90.653;
   1:  PR[91,2] = PR[90,2] + -8.202;
   1:  PR[91,3] = PR[90,3] + 145.128;
   1:L PR[91] R[100]mm/sec CNT100;
   1:  PR[91,1] = PR[90,1] + 90.681;
   1:  PR[91,2] = PR[90,2] + -7.857;
   1:  PR[91,3] = PR[90,3] + 145.129;
   1:L PR[91] R[100]mm/sec CNT100;
   1:  PR[91,1] = PR[90,1] + 91.700;
   1:  PR[91,2] = PR[90,2] + -0.670;
   1:  PR[91,3] = PR[90,3] + 145.131;
   1:L PR[91] R[100]mm/sec CNT100;
   1:  PR[91,1] = PR[90,1] + 91.686;
   1:  PR[91,2] = PR[90,2] + -0.501;
   1:  PR[91,3] = PR[90,3] + 145.172;
   1:L PR[91] R[100]mm/sec CNT100;
   1:  PR[91,1] = PR[90,1] + 90.667;
   1:  PR[91,2] = PR[90,2] + 6.686;
   1:  PR[91,3] = PR[90,3] + 145.173;
   1:L PR[91] R[100]mm/sec CNT100;
   1:  PR[91,1] = PR[90,1] + 90.619;
   1:  PR[91,2] = PR[90,2] + 6.877;
   1:  PR[91,3] = PR[90,3] + 145.214;
   1:L PR[91] R[100]mm/sec CNT100;
   1:  PR[91,1] = PR[90,1] + 90.500;
   1:  PR[91,2] = PR[90,2] + 7.159;
   1:  PR[91,3] = PR[90,3] + 145.215;
   1:L PR[91] R[100]mm/sec CNT100;
   1:  PR[91,1] = PR[90,1] + 87.388;
   1:  PR[91,2] = PR[90,2] + 14.125;
   1:  PR[91,3] = PR[90,3] + 145.217;
   1:L PR[91] R[100]mm/sec CNT100;
   1:  PR[91,1] = PR[90,1] + 87.269;
   1:  PR[91,2] = PR[90,2] + 14.317;
   1:  PR[91,3] = PR[90,3] + 145.260;
   1:L PR[91] R[100]mm/sec CNT100;
   1:  PR[91,1] = PR[90,1] + 81.705;
   1:  PR[91,2] = PR[90,2] + 21.030;
   1:  PR[91,3] = PR[90,3] + 145.261;
   1:L PR[91] R[100]mm/sec CNT100;
   1:  PR[91,1] = PR[90,1] + 81.473;
   1:  PR[91,2] = PR[90,2] + 21.238;
   1:  PR[91,3] = PR[90,3] + 145.310;
   1:L PR[91] R[100]mm/sec CNT100;
   1:  PR[91,1] = PR[90,1] + 73.585;
   1:  PR[91,2] = PR[90,2] + 26.830;
   1:  PR[91,3] = PR[90,3] + 145.312;
   1:L PR[91] R[100]mm/sec CNT100;
   1:  PR[91,1] = PR[90,1] + 73.200;
   1:  PR[91,2] = PR[90,2] + 27.027;
   1:  PR[91,3] = PR[90,3] + 145.367;
   1:L PR[91] R[100]mm/sec CNT100;
   1:  PR[91,1] = PR[90,1] + 63.360;
   1:  PR[91,2] = PR[90,2] + 30.787;
   1:  PR[91,3] = PR[90,3] + 145.369;
   1:L PR[91] R[100]mm/sec CNT100;
   1:  PR[91,1] = PR[90,1] + 62.732;
   1:  PR[91,2] = PR[90,2] + 30.938;
   1:  PR[91,3] = PR[90,3] + 145.429;
   1:L PR[91] R[100]mm/sec CNT100;
   1:  PR[91,1] = PR[90,1] + 57.788;
   1:  PR[91,2] = PR[90,2] + 31.850;
   1:  PR[91,3] = PR[90,3] + 145.432;
   1:L PR[91] R[100]mm/sec CNT100;
   1:  PR[91,1] = PR[90,1] + 56.998;
   1:  PR[91,2] = PR[90,2] + 31.946;
   1:  PR[91,3] = PR[90,3] + 145.461;
   1:L PR[91] R[100]mm/sec CNT100;
   1:  PR[91,1] = PR[90,1] + 52.000;
   1:  PR[91,2] = PR[90,2] + 32.252;
   1:  PR[91,3] = PR[90,3] + 145.465;
   1:L PR[91] R[100]mm/sec CNT100;
   1:  PR[91,1] = PR[90,1] + 51.100;
   1:  PR[91,2] = PR[90,2] + 32.260;
   1:  PR[91,3] = PR[90,3] + 145.493;
   1:L PR[91] R[100]mm/sec CNT100;
   1:  PR[91,1] = PR[90,1] + 46.236;
   1:  PR[91,2] = PR[90,2] + 31.962;
   1:  PR[91,3] = PR[90,3] + 145.499;
   1:L PR[91] R[100]mm/sec CNT100;
   1:  PR[91,1] = PR[90,1] + 45.294;
   1:  PR[91,2] = PR[90,2] + 31.868;
   1:  PR[91,3] = PR[90,3] + 145.526;
   1:L PR[91] R[100]mm/sec CNT100;
   1:  PR[91,1] = PR[90,1] + 40.744;
   1:  PR[91,2] = PR[90,2] + 31.028;
   1:  PR[91,3] = PR[90,3] + 145.531;
   1:L PR[91] R[100]mm/sec CNT100;
   1:  PR[91,1] = PR[90,1] + 39.708;
   1:  PR[91,2] = PR[90,2] + 30.814;
   1:  PR[91,3] = PR[90,3] + 145.558;
   1:L PR[91] R[100]mm/sec CNT100;
   1:  PR[91,1] = PR[90,1] + 38.373;
   1:  PR[91,2] = PR[90,2] + 30.386;
   1:  PR[91,3] = PR[90,3] + 145.564;
   1:L PR[91] R[100]mm/sec CNT100;
   1:  PR[91,1] = PR[90,1] + 36.383;
   1:  PR[91,2] = PR[90,2] + 29.538;
   1:  PR[91,3] = PR[90,3] + 145.571;
   1:L PR[91] R[100]mm/sec CNT100;
   1:  PR[91,1] = PR[90,1] + 29.629;
   1:  PR[91,2] = PR[90,2] + 26.952;
   1:  PR[91,3] = PR[90,3] + 145.584;
   1:L PR[91] R[100]mm/sec CNT100;
   1:  PR[91,1] = PR[90,1] + 27.969;
   1:  PR[91,2] = PR[90,2] + 25.961;
   1:  PR[91,3] = PR[90,3] + 145.625;
   1:L PR[91] R[100]mm/sec CNT100;
   1:  PR[91,1] = PR[90,1] + 25.362;
   1:  PR[91,2] = PR[90,2] + 24.026;
   1:  PR[91,3] = PR[90,3] + 145.635;
   1:L PR[91] R[100]mm/sec CNT100;
   1:  PR[91,1] = PR[90,1] + 21.771;
   1:  PR[91,2] = PR[90,2] + 21.475;
   1:  PR[91,3] = PR[90,3] + 145.654;
   1:L PR[91] R[100]mm/sec CNT100;
   1:  PR[91,1] = PR[90,1] + 19.587;
   1:  PR[91,2] = PR[90,2] + 19.291;
   1:  PR[91,3] = PR[90,3] + 145.679;
   1:L PR[91] R[100]mm/sec CNT100;
   1:  PR[91,1] = PR[90,1] + 16.214;
   1:  PR[91,2] = PR[90,2] + 15.087;
   1:  PR[91,3] = PR[90,3] + 145.696;
   1:L PR[91] R[100]mm/sec CNT100;
   1:  PR[91,1] = PR[90,1] + 14.004;
   1:  PR[91,2] = PR[90,2] + 11.167;
   1:  PR[91,3] = PR[90,3] + 145.727;
   1:L PR[91] R[100]mm/sec CNT100;
   1:  PR[91,1] = PR[90,1] + 12.824;
   1:  PR[91,2] = PR[90,2] + 8.174;
   1:  PR[91,3] = PR[90,3] + 145.752;
   1:L PR[91] R[100]mm/sec CNT100;
   1:  PR[91,1] = PR[90,1] + 12.336;
   1:  PR[91,2] = PR[90,2] + 6.626;
   1:  PR[91,3] = PR[90,3] + 145.770;
   1:L PR[91] R[100]mm/sec CNT100;
   1:  PR[91,1] = PR[90,1] + 11.712;
   1:  PR[91,2] = PR[90,2] + 3.932;
   1:  PR[91,3] = PR[90,3] + 145.779;
   1:L PR[91] R[100]mm/sec CNT100;
   1:  PR[91] = PR[90];
   1:  PR[91,1] = PR[90,1] + 12.432;
   1:  PR[91,2] = PR[90,2] + 2.781;
   1:  PR[91,3] = PR[90,3] + 147.095;
   1:L PR[91] R[100]mm/sec CNT100;
   1:  PR[91,1] = PR[90,1] + 12.168;
   1:  PR[91,2] = PR[90,2] + -0.700;
   1:  PR[91,3] = PR[90,3] + 145.800;
   1:L PR[91] R[100]mm/sec CNT100;
   1:  PR[91,1] = PR[90,1] + 12.265;
   1:  PR[91,2] = PR[90,2] + -1.617;
   1:  PR[91,3] = PR[90,3] + 145.819;
   1:L PR[91] R[100]mm/sec CNT100;
   1:  PR[91,1] = PR[90,1] + 12.524;
   1:  PR[91,2] = PR[90,2] + -5.080;
   1:  PR[91,3] = PR[90,3] + 145.825;
   1:L PR[91] R[100]mm/sec CNT100;
   1:  PR[91,1] = PR[90,1] + 13.363;
   1:  PR[91,2] = PR[90,2] + -8.701;
   1:  PR[91,3] = PR[90,3] + 145.844;
   1:L PR[91] R[100]mm/sec CNT100;
   1:  PR[91,1] = PR[90,1] + 13.467;
   1:  PR[91,2] = PR[90,2] + -9.033;
   1:  PR[91,3] = PR[90,3] + 145.865;
   1:L PR[91] R[100]mm/sec CNT100;
   1:  PR[91,1] = PR[90,1] + 14.443;
   1:  PR[91,2] = PR[90,2] + -11.507;
   1:  PR[91,3] = PR[90,3] + 145.867;
   1:L PR[91] R[100]mm/sec CNT100;
   1:  PR[91,1] = PR[90,1] + 14.819;
   1:  PR[91,2] = PR[90,2] + -12.449;
   1:  PR[91,3] = PR[90,3] + 145.882;
   1:L PR[91] R[100]mm/sec CNT100;
   1:  PR[91,1] = PR[90,1] + 15.091;
   1:  PR[91,2] = PR[90,2] + -13.057;
   1:  PR[91,3] = PR[90,3] + 145.888;
   1:L PR[91] R[100]mm/sec CNT100;
   1:  PR[91,1] = PR[90,1] + 16.893;
   1:  PR[91,2] = PR[90,2] + -16.241;
   1:  PR[91,3] = PR[90,3] + 145.892;
   1:L PR[91] R[100]mm/sec CNT100;
   1:  PR[91,1] = PR[90,1] + 18.093;
   1:  PR[91,2] = PR[90,2] + -17.774;
   1:  PR[91,3] = PR[90,3] + 145.912;
   1:L PR[91] R[100]mm/sec CNT100;
   1:  PR[91,1] = PR[90,1] + 21.090;
   1:  PR[91,2] = PR[90,2] + -21.393;
   1:  PR[91,3] = PR[90,3] + 145.923;
   1:L PR[91] R[100]mm/sec CNT100;
   1:  PR[91,1] = PR[90,1] + 22.507;
   1:  PR[91,2] = PR[90,2] + -22.809;
   1:  PR[91,3] = PR[90,3] + 145.950;
   1:L PR[91] R[100]mm/sec CNT100;
   1:  PR[91,1] = PR[90,1] + 23.466;
   1:  PR[91,2] = PR[90,2] + -23.539;
   1:  PR[91,3] = PR[90,3] + 145.961;
   1:L PR[91] R[100]mm/sec CNT100;
   1:  PR[91,1] = PR[90,1] + 29.404;
   1:  PR[91,2] = PR[90,2] + -27.758;
   1:  PR[91,3] = PR[90,3] + 145.968;
   1:L PR[91] R[100]mm/sec CNT100;
   1:  PR[91,1] = PR[90,1] + 30.491;
   1:  PR[91,2] = PR[90,2] + -28.406;
   1:  PR[91,3] = PR[90,3] + 146.009;
   1:L PR[91] R[100]mm/sec CNT100;
   1:  PR[91,1] = PR[90,1] + 31.170;
   1:  PR[91,2] = PR[90,2] + -28.710;
   1:  PR[91,3] = PR[90,3] + 146.016;
   1:L PR[91] R[100]mm/sec CNT100;
   1:  PR[91,1] = PR[90,1] + 31.799;
   1:  PR[91,2] = PR[90,2] + -28.892;
   1:  PR[91,3] = PR[90,3] + 146.021;
   1:L PR[91] R[100]mm/sec CNT100;
   1:  PR[91,1] = PR[90,1] + 40.698;
   1:  PR[91,2] = PR[90,2] + -32.299;
   1:  PR[91,3] = PR[90,3] + 146.024;
   1:L PR[91] R[100]mm/sec CNT100;
   1:  PR[91,1] = PR[90,1] + 41.288;
   1:  PR[91,2] = PR[90,2] + -32.421;
   1:  PR[91,3] = PR[90,3] + 146.078;
   1:L PR[91] R[100]mm/sec CNT100;
   1:  PR[91,1] = PR[90,1] + 46.282;
   1:  PR[91,2] = PR[90,2] + -33.342;
   1:  PR[91,3] = PR[90,3] + 146.081;
   1:L PR[91] R[100]mm/sec CNT100;
   1:  PR[91,1] = PR[90,1] + 46.866;
   1:  PR[91,2] = PR[90,2] + -33.400;
   1:  PR[91,3] = PR[90,3] + 146.110;
   1:L PR[91] R[100]mm/sec CNT100;
   1:  PR[91,1] = PR[90,1] + 52.131;
   1:  PR[91,2] = PR[90,2] + -33.722;
   1:  PR[91,3] = PR[90,3] + 146.113;
   1:L PR[91] R[100]mm/sec CNT100;
   1:  PR[91,1] = PR[90,1] + 52.686;
   1:  PR[91,2] = PR[90,2] + -33.717;
   1:  PR[91,3] = PR[90,3] + 146.143;
   1:L PR[91] R[100]mm/sec CNT100;
   1:  PR[91,1] = PR[90,1] + 58.040;
   1:  PR[91,2] = PR[90,2] + -33.389;
   1:  PR[91,3] = PR[90,3] + 146.146;
   1:L PR[91] R[100]mm/sec CNT100;
   1:  PR[91,1] = PR[90,1] + 58.523;
   1:  PR[91,2] = PR[90,2] + -33.330;
   1:  PR[91,3] = PR[90,3] + 146.177;
   1:L PR[91] R[100]mm/sec CNT100;
   1:  PR[91,1] = PR[90,1] + 63.775;
   1:  PR[91,2] = PR[90,2] + -32.361;
   1:  PR[91,3] = PR[90,3] + 146.179;
   1:L PR[91] R[100]mm/sec CNT100;
   1:  PR[91,1] = PR[90,1] + 64.140;
   1:  PR[91,2] = PR[90,2] + -32.273;
   1:  PR[91,3] = PR[90,3] + 146.210;
   1:L PR[91] R[100]mm/sec CNT100;
   1:  PR[91,1] = PR[90,1] + 64.443;
   1:  PR[91,2] = PR[90,2] + -32.160;
   1:  PR[91,3] = PR[90,3] + 146.212;
   1:L PR[91] R[100]mm/sec CNT100;
   1:  PR[91,1] = PR[90,1] + 74.220;
   1:  PR[91,2] = PR[90,2] + -28.416;
   1:  PR[91,3] = PR[90,3] + 146.214;
   1:L PR[91] R[100]mm/sec CNT100;
   1:  PR[91,1] = PR[90,1] + 74.399;
   1:  PR[91,2] = PR[90,2] + -28.324;
   1:  PR[91,3] = PR[90,3] + 146.273;
   1:L PR[91] R[100]mm/sec CNT100;
   1:  PR[91,1] = PR[90,1] + 82.448;
   1:  PR[91,2] = PR[90,2] + -22.613;
   1:  PR[91,3] = PR[90,3] + 146.274;
   1:L PR[91] R[100]mm/sec CNT100;
   1:  PR[91,1] = PR[90,1] + 82.536;
   1:  PR[91,2] = PR[90,2] + -22.534;
   1:  PR[91,3] = PR[90,3] + 146.330;
   1:L PR[91] R[100]mm/sec CNT100;
   1:  PR[91,1] = PR[90,1] + 88.194;
   1:  PR[91,2] = PR[90,2] + -15.703;
   1:L PR[91] R[100]mm/sec CNT100;
   1:  PR[91,1] = PR[90,1] + 88.225;
   1:  PR[91,2] = PR[90,2] + -15.655;
   1:  PR[91,3] = PR[90,3] + 146.380;
   1:L PR[91] R[100]mm/sec CNT100;
   1:  PR[91,1] = PR[90,1] + 91.506;
   1:  PR[91,2] = PR[90,2] + -8.293;
   1:  PR[91,3] = PR[90,3] + 146.381;
   1:L PR[91] R[100]mm/sec CNT100;
   1:  PR[91,1] = PR[90,1] + 91.521;
   1:  PR[91,2] = PR[90,2] + -8.118;
   1:  PR[91,3] = PR[90,3] + 146.426;
   1:L PR[91] R[100]mm/sec CNT100;
   1:  PR[91,1] = PR[90,1] + 92.577;
   1:  PR[91,2] = PR[90,2] + -0.670;
   1:  PR[91,3] = PR[90,3] + 146.427;
   1:L PR[91] R[100]mm/sec CNT100;
   1:  PR[91,1] = PR[90,1] + 92.575;
   1:  PR[91,2] = PR[90,2] + -0.653;
   1:  PR[91,3] = PR[90,3] + 146.470;
   1:L PR[91] R[100]mm/sec CNT100;
   1:  PR[91,1] = PR[90,1] + 91.519;
   1:  PR[91,2] = PR[90,2] + 6.795;
   1:L PR[91] R[100]mm/sec CNT100;
   1:  PR[91,1] = PR[90,1] + 91.509;
   1:  PR[91,2] = PR[90,2] + 6.837;
   1:  PR[91,3] = PR[90,3] + 146.512;
   1:L PR[91] R[100]mm/sec CNT100;
   1:  PR[91,1] = PR[90,1] + 91.453;
   1:  PR[91,2] = PR[90,2] + 6.969;
   1:  PR[91,3] = PR[90,3] + 146.513;
   1:L PR[91] R[100]mm/sec CNT100;
   1:  PR[91,1] = PR[90,1] + 88.223;
   1:  PR[91,2] = PR[90,2] + 14.198;
   1:L PR[91] R[100]mm/sec CNT100;
   1:  PR[91,1] = PR[90,1] + 88.193;
   1:  PR[91,2] = PR[90,2] + 14.247;
   1:  PR[91,3] = PR[90,3] + 146.558;
   1:L PR[91] R[100]mm/sec CNT100;
   1:  PR[91,1] = PR[90,1] + 82.532;
   1:  PR[91,2] = PR[90,2] + 21.079;
   1:  PR[91,3] = PR[90,3] + 146.559;
   1:L PR[91] R[100]mm/sec CNT100;
   1:  PR[91,1] = PR[90,1] + 82.444;
   1:  PR[91,2] = PR[90,2] + 21.157;
   1:  PR[91,3] = PR[90,3] + 146.609;
   1:L PR[91] R[100]mm/sec CNT100;
   1:  PR[91,1] = PR[90,1] + 74.394;
   1:  PR[91,2] = PR[90,2] + 26.868;
   1:L PR[91] R[100]mm/sec CNT100;
   1:  PR[91,1] = PR[90,1] + 74.216;
   1:  PR[91,2] = PR[90,2] + 26.960;
   1:  PR[91,3] = PR[90,3] + 146.665;
   1:L PR[91] R[100]mm/sec CNT100;
   1:  PR[91,1] = PR[90,1] + 64.126;
   1:  PR[91,2] = PR[90,2] + 30.818;
   1:  PR[91,3] = PR[90,3] + 146.666;
   1:L PR[91] R[100]mm/sec CNT100;
   1:  PR[91,1] = PR[90,1] + 63.770;
   1:  PR[91,2] = PR[90,2] + 30.903;
   1:  PR[91,3] = PR[90,3] + 146.727;
   1:L PR[91] R[100]mm/sec CNT100;
   1:  PR[91,1] = PR[90,1] + 58.518;
   1:  PR[91,2] = PR[90,2] + 31.872;
   1:  PR[91,3] = PR[90,3] + 146.729;
   1:L PR[91] R[100]mm/sec CNT100;
   1:  PR[91,1] = PR[90,1] + 58.035;
   1:  PR[91,2] = PR[90,2] + 31.931;
   1:  PR[91,3] = PR[90,3] + 146.760;
   1:L PR[91] R[100]mm/sec CNT100;
   1:  PR[91,1] = PR[90,1] + 52.681;
   1:  PR[91,2] = PR[90,2] + 32.258;
   1:  PR[91,3] = PR[90,3] + 146.762;
   1:L PR[91] R[100]mm/sec CNT100;
   1:  PR[91,1] = PR[90,1] + 52.126;
   1:  PR[91,2] = PR[90,2] + 32.263;
   1:  PR[91,3] = PR[90,3] + 146.793;
   1:L PR[91] R[100]mm/sec CNT100;
   1:  PR[91,1] = PR[90,1] + 46.860;
   1:  PR[91,2] = PR[90,2] + 31.941;
   1:  PR[91,3] = PR[90,3] + 146.796;
   1:L PR[91] R[100]mm/sec CNT100;
   1:  PR[91,1] = PR[90,1] + 46.277;
   1:  PR[91,2] = PR[90,2] + 31.883;
   1:  PR[91,3] = PR[90,3] + 146.826;
   1:L PR[91] R[100]mm/sec CNT100;
   1:  PR[91,1] = PR[90,1] + 41.284;
   1:  PR[91,2] = PR[90,2] + 30.961;
   1:  PR[91,3] = PR[90,3] + 146.829;
   1:L PR[91] R[100]mm/sec CNT100;
   1:  PR[91,1] = PR[90,1] + 40.638;
   1:  PR[91,2] = PR[90,2] + 30.827;
   1:  PR[91,3] = PR[90,3] + 146.858;
   1:L PR[91] R[100]mm/sec CNT100;
   1:  PR[91,1] = PR[90,1] + 39.818;
   1:  PR[91,2] = PR[90,2] + 30.564;
   1:  PR[91,3] = PR[90,3] + 146.861;
   1:L PR[91] R[100]mm/sec CNT100;
   1:  PR[91,1] = PR[90,1] + 38.516;
   1:  PR[91,2] = PR[90,2] + 30.010;
   1:  PR[91,3] = PR[90,3] + 146.866;
   1:L PR[91] R[100]mm/sec CNT100;
   1:  PR[91,1] = PR[90,1] + 30.440;
   1:  PR[91,2] = PR[90,2] + 26.917;
   1:  PR[91,3] = PR[90,3] + 146.874;
   1:L PR[91] R[100]mm/sec CNT100;
   1:  PR[91,1] = PR[90,1] + 29.419;
   1:  PR[91,2] = PR[90,2] + 26.308;
   1:  PR[91,3] = PR[90,3] + 146.923;
   1:L PR[91] R[100]mm/sec CNT100;
   1:  PR[91,1] = PR[90,1] + 27.713;
   1:  PR[91,2] = PR[90,2] + 25.041;
   1:  PR[91,3] = PR[90,3] + 146.930;
   1:L PR[91] R[100]mm/sec CNT100;
   1:  PR[91,1] = PR[90,1] + 22.481;
   1:  PR[91,2] = PR[90,2] + 21.324;
   1:  PR[91,3] = PR[90,3] + 146.942;
   1:L PR[91] R[100]mm/sec CNT100;
   1:  PR[91,1] = PR[90,1] + 21.099;
   1:  PR[91,2] = PR[90,2] + 19.943;
   1:  PR[91,3] = PR[90,3] + 146.978;
   1:L PR[91] R[100]mm/sec CNT100;
   1:  PR[91,1] = PR[90,1] + 18.830;
   1:  PR[91,2] = PR[90,2] + 17.114;
   1:  PR[91,3] = PR[90,3] + 146.989;
   1:L PR[91] R[100]mm/sec CNT100;
   1:  PR[91,1] = PR[90,1] + 16.879;
   1:  PR[91,2] = PR[90,2] + 14.757;
   1:  PR[91,3] = PR[90,3] + 147.010;
   1:L PR[91] R[100]mm/sec CNT100;
   1:  PR[91,1] = PR[90,1] + 15.102;
   1:  PR[91,2] = PR[90,2] + 11.618;
   1:  PR[91,3] = PR[90,3] + 147.027;
   1:L PR[91] R[100]mm/sec CNT100;
   1:  PR[91,1] = PR[90,1] + 14.436;
   1:  PR[91,2] = PR[90,2] + 10.031;
   1:  PR[91,3] = PR[90,3] + 147.047;
   1:L PR[91] R[100]mm/sec CNT100;
   1:  PR[91,1] = PR[90,1] + 13.467;
   1:  PR[91,2] = PR[90,2] + 7.575;
   1:  PR[91,3] = PR[90,3] + 147.057;
   1:L PR[91] R[100]mm/sec CNT100;
   1:  PR[91,1] = PR[90,1] + 13.363;
   1:  PR[91,2] = PR[90,2] + 7.242;
   1:  PR[91,3] = PR[90,3] + 147.072;
   1:L PR[91] R[100]mm/sec CNT100;
   1:  PR[91,1] = PR[90,1] + 12.517;
   1:  PR[91,2] = PR[90,2] + 3.592;
   1:  PR[91,3] = PR[90,3] + 147.074;
   1:L PR[91] R[100]mm/sec CNT100;
   1:  PR[91] = PR[90];
   1:  PR[91,1] = PR[90,1] + 13.157;
   1:  PR[91,2] = PR[90,2] + 0.028;
   1:  PR[91,3] = PR[90,3] + 148.395;
   1:L PR[91] R[100]mm/sec CNT100;
   1:  PR[91,1] = PR[90,1] + 13.041;
   1:  PR[91,2] = PR[90,2] + -0.795;
   1:  PR[91,3] = PR[90,3] + 147.118;
   1:L PR[91] R[100]mm/sec CNT100;
   1:  PR[91,1] = PR[90,1] + 13.285;
   1:  PR[91,2] = PR[90,2] + -3.999;
   1:  PR[91,3] = PR[90,3] + 147.123;
   1:L PR[91] R[100]mm/sec CNT100;
   1:  PR[91,1] = PR[90,1] + 13.502;
   1:  PR[91,2] = PR[90,2] + -5.536;
   1:  PR[91,3] = PR[90,3] + 147.141;
   1:L PR[91] R[100]mm/sec CNT100;
   1:  PR[91,1] = PR[90,1] + 14.210;
   1:  PR[91,2] = PR[90,2] + -8.632;
   1:  PR[91,3] = PR[90,3] + 147.150;
   1:L PR[91] R[100]mm/sec CNT100;
   1:  PR[91,1] = PR[90,1] + 14.845;
   1:  PR[91,2] = PR[90,2] + -10.222;
   1:  PR[91,3] = PR[90,3] + 147.168;
   1:L PR[91] R[100]mm/sec CNT100;
   1:  PR[91,1] = PR[90,1] + 16.743;
   1:  PR[91,2] = PR[90,2] + -14.471;
   1:  PR[91,3] = PR[90,3] + 147.178;
   1:L PR[91] R[100]mm/sec CNT100;
   1:  PR[91,1] = PR[90,1] + 17.567;
   1:  PR[91,2] = PR[90,2] + -15.926;
   1:  PR[91,3] = PR[90,3] + 147.204;
   1:L PR[91] R[100]mm/sec CNT100;
   1:  PR[91,1] = PR[90,1] + 18.101;
   1:  PR[91,2] = PR[90,2] + -16.609;
   1:  PR[91,3] = PR[90,3] + 147.213;
   1:L PR[91] R[100]mm/sec CNT100;
   1:  PR[91,1] = PR[90,1] + 22.604;
   1:  PR[91,2] = PR[90,2] + -22.045;
   1:  PR[91,3] = PR[90,3] + 147.218;
   1:L PR[91] R[100]mm/sec CNT100;
   1:  PR[91,1] = PR[90,1] + 23.218;
   1:  PR[91,2] = PR[90,2] + -22.659;
   1:  PR[91,3] = PR[90,3] + 147.258;
   1:L PR[91] R[100]mm/sec CNT100;
   1:  PR[91,1] = PR[90,1] + 23.621;
   1:  PR[91,2] = PR[90,2] + -22.966;
   1:  PR[91,3] = PR[90,3] + 147.263;
   1:L PR[91] R[100]mm/sec CNT100;
   1:  PR[91,1] = PR[90,1] + 30.855;
   1:  PR[91,2] = PR[90,2] + -28.104;
   1:  PR[91,3] = PR[90,3] + 147.266;
   1:L PR[91] R[100]mm/sec CNT100;
   1:  PR[91,1] = PR[90,1] + 31.302;
   1:  PR[91,2] = PR[90,2] + -28.371;
   1:  PR[91,3] = PR[90,3] + 147.316;
   1:L PR[91] R[100]mm/sec CNT100;
   1:  PR[91,1] = PR[90,1] + 31.517;
   1:  PR[91,2] = PR[90,2] + -28.467;
   1:  PR[91,3] = PR[90,3] + 147.319;
   1:L PR[91] R[100]mm/sec CNT100;
   1:  PR[91,1] = PR[90,1] + 31.799;
   1:  PR[91,2] = PR[90,2] + -28.549;
   1:  PR[91,3] = PR[90,3] + 147.320;
   1:L PR[91] R[100]mm/sec CNT100;
   1:  PR[91,1] = PR[90,1] + 41.610;
   1:  PR[91,2] = PR[90,2] + -32.305;
   1:  PR[91,3] = PR[90,3] + 147.322;
   1:L PR[91] R[100]mm/sec CNT100;
   1:  PR[91,1] = PR[90,1] + 47.267;
   1:  PR[91,2] = PR[90,2] + -33.357;
   1:  PR[91,3] = PR[90,3] + 147.381;
   1:L PR[91] R[100]mm/sec CNT100;
   1:  PR[91,1] = PR[90,1] + 47.490;
   1:  PR[91,2] = PR[90,2] + -33.379;
   1:  PR[91,3] = PR[90,3] + 147.414;
   1:L PR[91] R[100]mm/sec CNT100;
   1:  PR[91,1] = PR[90,1] + 53.158;
   1:  PR[91,2] = PR[90,2] + -33.726;
   1:  PR[91,3] = PR[90,3] + 147.415;
   1:L PR[91] R[100]mm/sec CNT100;
   1:  PR[91,1] = PR[90,1] + 53.368;
   1:  PR[91,2] = PR[90,2] + -33.724;
   1:  PR[91,3] = PR[90,3] + 147.447;
   1:L PR[91] R[100]mm/sec CNT100;
   1:  PR[91,1] = PR[90,1] + 59.077;
   1:  PR[91,2] = PR[90,2] + -33.374;
   1:  PR[91,3] = PR[90,3] + 147.448;
   1:L PR[91] R[100]mm/sec CNT100;
   1:  PR[91,1] = PR[90,1] + 59.253;
   1:  PR[91,2] = PR[90,2] + -33.352;
   1:  PR[91,3] = PR[90,3] + 147.481;
   1:L PR[91] R[100]mm/sec CNT100;
   1:  PR[91,1] = PR[90,1] + 64.813;
   1:  PR[91,2] = PR[90,2] + -32.326;
   1:  PR[91,3] = PR[90,3] + 147.482;
   1:L PR[91] R[100]mm/sec CNT100;
   1:  PR[91,1] = PR[90,1] + 64.906;
   1:  PR[91,2] = PR[90,2] + -32.304;
   1:  PR[91,3] = PR[90,3] + 147.514;
   1:L PR[91] R[100]mm/sec CNT100;
   1:  PR[91,1] = PR[90,1] + 64.993;
   1:  PR[91,2] = PR[90,2] + -32.271;
   1:L PR[91] R[100]mm/sec CNT100;
   1:  PR[91,1] = PR[90,1] + 75.220;
   1:  PR[91,2] = PR[90,2] + -28.355;
   1:  PR[91,3] = PR[90,3] + 147.515;
   1:L PR[91] R[100]mm/sec CNT100;
   1:  PR[91,1] = PR[90,1] + 83.384;
   1:  PR[91,2] = PR[90,2] + -22.557;
   1:  PR[91,3] = PR[90,3] + 147.577;
   1:L PR[91] R[100]mm/sec CNT100;
   1:  PR[91,1] = PR[90,1] + 89.083;
   1:  PR[91,2] = PR[90,2] + -15.676;
   1:  PR[91,3] = PR[90,3] + 147.633;
   1:L PR[91] R[100]mm/sec CNT100;
   1:  PR[91,1] = PR[90,1] + 92.383;
   1:  PR[91,2] = PR[90,2] + -8.281;
   1:  PR[91,3] = PR[90,3] + 147.684;
   1:L PR[91] R[100]mm/sec CNT100;
   1:  PR[91,1] = PR[90,1] + 93.446;
   1:  PR[91,2] = PR[90,2] + -0.729;
   1:  PR[91,3] = PR[90,3] + 147.730;
   1:L PR[91] R[100]mm/sec CNT100;
   1:  PR[91,1] = PR[90,1] + 92.381;
   1:  PR[91,2] = PR[90,2] + 6.834;
   1:  PR[91,3] = PR[90,3] + 147.773;
   1:L PR[91] R[100]mm/sec CNT100;
   1:  PR[91,1] = PR[90,1] + 89.082;
   1:  PR[91,2] = PR[90,2] + 14.219;
   1:  PR[91,3] = PR[90,3] + 147.816;
   1:L PR[91] R[100]mm/sec CNT100;
   1:  PR[91,1] = PR[90,1] + 83.380;
   1:  PR[91,2] = PR[90,2] + 21.102;
   1:  PR[91,3] = PR[90,3] + 147.861;
   1:L PR[91] R[100]mm/sec CNT100;
   1:  PR[91,1] = PR[90,1] + 75.215;
   1:  PR[91,2] = PR[90,2] + 26.899;
   1:  PR[91,3] = PR[90,3] + 147.912;
   1:L PR[91] R[100]mm/sec CNT100;
   1:  PR[91,1] = PR[90,1] + 64.892;
   1:  PR[91,2] = PR[90,2] + 30.848;
   1:  PR[91,3] = PR[90,3] + 147.969;
   1:L PR[91] R[100]mm/sec CNT100;
   1:  PR[91,1] = PR[90,1] + 64.807;
   1:  PR[91,2] = PR[90,2] + 30.868;
   1:  PR[91,3] = PR[90,3] + 148.031;
   1:L PR[91] R[100]mm/sec CNT100;
   1:  PR[91,1] = PR[90,1] + 59.247;
   1:  PR[91,2] = PR[90,2] + 31.894;
   1:  PR[91,3] = PR[90,3] + 148.032;
   1:L PR[91] R[100]mm/sec CNT100;
   1:  PR[91,1] = PR[90,1] + 59.072;
   1:  PR[91,2] = PR[90,2] + 31.916;
   1:  PR[91,3] = PR[90,3] + 148.064;
   1:L PR[91] R[100]mm/sec CNT100;
   1:  PR[91,1] = PR[90,1] + 53.363;
   1:  PR[91,2] = PR[90,2] + 32.265;
   1:  PR[91,3] = PR[90,3] + 148.065;
   1:L PR[91] R[100]mm/sec CNT100;
   1:  PR[91,1] = PR[90,1] + 53.153;
   1:  PR[91,2] = PR[90,2] + 32.267;
   1:  PR[91,3] = PR[90,3] + 148.097;
   1:L PR[91] R[100]mm/sec CNT100;
   1:  PR[91,1] = PR[90,1] + 47.485;
   1:  PR[91,2] = PR[90,2] + 31.919;
   1:  PR[91,3] = PR[90,3] + 148.098;
   1:L PR[91] R[100]mm/sec CNT100;
   1:  PR[91,1] = PR[90,1] + 47.260;
   1:  PR[91,2] = PR[90,2] + 31.897;
   1:  PR[91,3] = PR[90,3] + 148.130;
   1:L PR[91] R[100]mm/sec CNT100;
   1:  PR[91,1] = PR[90,1] + 41.822;
   1:  PR[91,2] = PR[90,2] + 30.893;
   1:  PR[91,3] = PR[90,3] + 148.131;
   1:L PR[91] R[100]mm/sec CNT100;
   1:  PR[91,1] = PR[90,1] + 41.569;
   1:  PR[91,2] = PR[90,2] + 30.841;
   1:  PR[91,3] = PR[90,3] + 148.163;
   1:L PR[91] R[100]mm/sec CNT100;
   1:  PR[91,1] = PR[90,1] + 41.262;
   1:  PR[91,2] = PR[90,2] + 30.742;
   1:  PR[91,3] = PR[90,3] + 148.164;
   1:L PR[91] R[100]mm/sec CNT100;
   1:  PR[91,1] = PR[90,1] + 40.649;
   1:  PR[91,2] = PR[90,2] + 30.481;
   1:  PR[91,3] = PR[90,3] + 148.166;
   1:L PR[91] R[100]mm/sec CNT100;
   1:  PR[91,1] = PR[90,1] + 31.250;
   1:  PR[91,2] = PR[90,2] + 26.882;
   1:  PR[91,3] = PR[90,3] + 148.170;
   1:L PR[91] R[100]mm/sec CNT100;
   1:  PR[91,1] = PR[90,1] + 30.868;
   1:  PR[91,2] = PR[90,2] + 26.654;
   1:  PR[91,3] = PR[90,3] + 148.227;
   1:L PR[91] R[100]mm/sec CNT100;
   1:  PR[91,1] = PR[90,1] + 30.063;
   1:  PR[91,2] = PR[90,2] + 26.056;
   1:  PR[91,3] = PR[90,3] + 148.229;
   1:L PR[91] R[100]mm/sec CNT100;
   1:  PR[91,1] = PR[90,1] + 23.191;
   1:  PR[91,2] = PR[90,2] + 21.173;
   1:  PR[91,3] = PR[90,3] + 148.235;
   1:L PR[91] R[100]mm/sec CNT100;
   1:  PR[91,1] = PR[90,1] + 22.612;
   1:  PR[91,2] = PR[90,2] + 20.595;
   1:  PR[91,3] = PR[90,3] + 148.282;
   1:L PR[91] R[100]mm/sec CNT100;
   1:  PR[91,1] = PR[90,1] + 21.528;
   1:  PR[91,2] = PR[90,2] + 19.243;
   1:  PR[91,3] = PR[90,3] + 148.287;
   1:L PR[91] R[100]mm/sec CNT100;
   1:  PR[91,1] = PR[90,1] + 17.552;
   1:  PR[91,2] = PR[90,2] + 14.442;
   1:  PR[91,3] = PR[90,3] + 148.297;
   1:L PR[91] R[100]mm/sec CNT100;
   1:  PR[91,1] = PR[90,1] + 16.754;
   1:  PR[91,2] = PR[90,2] + 13.031;
   1:  PR[91,3] = PR[90,3] + 148.332;
   1:L PR[91] R[100]mm/sec CNT100;
   1:  PR[91,1] = PR[90,1] + 15.495;
   1:  PR[91,2] = PR[90,2] + 10.029;
   1:  PR[91,3] = PR[90,3] + 148.341;
   1:L PR[91] R[100]mm/sec CNT100;
   1:  PR[91,1] = PR[90,1] + 14.201;
   1:  PR[91,2] = PR[90,2] + 7.134;
   1:  PR[91,3] = PR[90,3] + 148.360;
   1:L PR[91] R[100]mm/sec CNT100;
   1:  PR[91,1] = PR[90,1] + 13.515;
   1:  PR[91,2] = PR[90,2] + 4.130;
   1:  PR[91,3] = PR[90,3] + 148.378;
   1:L PR[91] R[100]mm/sec CNT100;
   1:  PR[91,1] = PR[90,1] + 13.157;
   1:  PR[91,2] = PR[90,2] + 0.028;
   1:  PR[91,3] = PR[90,3] + 148.395;
   1:L PR[91] R[100]mm/sec CNT100;
   1:  PR[91,1] = PR[90,1] + 13.041;
   1:  PR[91,2] = PR[90,2] + -0.795;
   1:L PR[91] R[100]mm/sec CNT100;
   1:  PR[91,1] = PR[90,1] + 13.285;
   1:  PR[91,2] = PR[90,2] + -3.999;
   1:L PR[91] R[100]mm/sec CNT100;
   1:  PR[91,1] = PR[90,1] + 13.502;
   1:  PR[91,2] = PR[90,2] + -5.536;
   1:L PR[91] R[100]mm/sec CNT100;
   1:  PR[91,1] = PR[90,1] + 14.210;
   1:  PR[91,2] = PR[90,2] + -8.632;
   1:L PR[91] R[100]mm/sec CNT100;
   1:  PR[91,1] = PR[90,1] + 14.845;
   1:  PR[91,2] = PR[90,2] + -10.222;
   1:L PR[91] R[100]mm/sec CNT100;
   1:  PR[91,1] = PR[90,1] + 16.743;
   1:  PR[91,2] = PR[90,2] + -14.471;
   1:L PR[91] R[100]mm/sec CNT100;
   1:  PR[91,1] = PR[90,1] + 17.567;
   1:  PR[91,2] = PR[90,2] + -15.926;
   1:L PR[91] R[100]mm/sec CNT100;
   1:  PR[91,1] = PR[90,1] + 18.101;
   1:  PR[91,2] = PR[90,2] + -16.609;
   1:L PR[91] R[100]mm/sec CNT100;
   1:  PR[91,1] = PR[90,1] + 22.604;
   1:  PR[91,2] = PR[90,2] + -22.045;
   1:L PR[91] R[100]mm/sec CNT100;
   1:  PR[91,1] = PR[90,1] + 23.218;
   1:  PR[91,2] = PR[90,2] + -22.659;
   1:L PR[91] R[100]mm/sec CNT100;
   1:  PR[91,1] = PR[90,1] + 23.621;
   1:  PR[91,2] = PR[90,2] + -22.966;
   1:L PR[91] R[100]mm/sec CNT100;
   1:  PR[91,1] = PR[90,1] + 30.855;
   1:  PR[91,2] = PR[90,2] + -28.104;
   1:L PR[91] R[100]mm/sec CNT100;
   1:  PR[91,1] = PR[90,1] + 31.302;
   1:  PR[91,2] = PR[90,2] + -28.371;
   1:L PR[91] R[100]mm/sec CNT100;
   1:  PR[91,1] = PR[90,1] + 31.517;
   1:  PR[91,2] = PR[90,2] + -28.467;
   1:L PR[91] R[100]mm/sec CNT100;
   1:  PR[91,1] = PR[90,1] + 31.799;
